# B&R Automation Studio project A2019059_Linka_Power_CP (part 36)

```iecst
            //Polohovanie na pozície skrutiek//
            IF P3_Srobovanie.RR_PolohujNaPoziciuSkrutky_4F5F THEN
                IF P3_Srobovanie.PAR.RR_IndexPozicieSkrutky_4F5F = 0 THEN  //Pozícia skrutky K40 a M5
                    SC_P3_Srobovanie.ResetStep:= TRUE;
                    SC_P3_Srobovanie.Step:= 170;
                ELSIF P3_Srobovanie.PAR.RR_IndexPozicieSkrutky_4F5F = 1 THEN  //Pozícia odobratia skrutky M5
                    SC_P3_Srobovanie.ResetStep:= TRUE;
                    SC_P3_Srobovanie.Step:= 130;
                ELSIF P3_Srobovanie.PAR.RR_IndexPozicieSkrutky_4F5F = 2 THEN  //Pozícia HV testu
                    SC_P3_Srobovanie.ResetStep:= TRUE;
                    SC_P3_Srobovanie.Step:= 300;
                END_IF
            ELSIF P3_Srobovanie.RR_PolohujNaPoziciuSkrutky_5H THEN
                IF P3_Srobovanie.PAR.RR_IndexPozicieSkrutky_5H = 0 THEN  //Pozícia skrutky M5
                    SC_P3_Srobovanie.ResetStep:= TRUE;
                    SC_P3_Srobovanie.Step:= 200;
                ELSIF P3_Srobovanie.PAR.RR_IndexPozicieSkrutky_5H = 1 THEN  //Pozícia odobratia skrutky M5
                    SC_P3_Srobovanie.ResetStep:= TRUE;
                    SC_P3_Srobovanie.Step:= 130;
                ELSIF P3_Srobovanie.PAR.RR_IndexPozicieSkrutky_5H = 2 THEN  //Pozícia HV testu
                    SC_P3_Srobovanie.ResetStep:= TRUE;
                    SC_P3_Srobovanie.Step:= 300;
                END_IF
            END_IF

    END_CASE

END_PROGRAM

PROGRAM _EXIT
	(* Insert code here *)

END_PROGRAM
```

#### Variables.var - Local variables
```iecst
VAR
	Triger_0 : BOOL;
	CasPowerON_OsY : TON;
	SC_OvlManipulatora_OsY : SequenceControlTyp;
	OsY_JoggVPRED : BOOL;
	OsY_JoggVZAD : BOOL;
	OsY_POLOHUJ : BOOL;
	OsY_HOME : BOOL;
	OsY_STOP : BOOL;
	ZadanaPoziciaUINT_OsY : UINT;
	AktualnaPoziciaUINT_OsY : UINT;
	SC_OvlZdvihuHV_Testu : SequenceControlTyp;
	HV_Test_VYSUN : BOOL;
	HV_Test_ZASUN : BOOL;
	SC_OvlKontaktovHV_Testu : SequenceControlTyp;
	Kontakty_VYSUN : BOOL;
	Kontakty_ZASUN : BOOL;
	SC_OvlTesteraHV : SequenceControlTyp;
	SKTcpClientTester_0 : SKTcpClientTester;
	dataStr : STRING[32];
	HV_Test_START : BOOL;
	HV_Test_UKONCENY : BOOL;
	i : USINT;
	CasSrobovania : REAL;
	M5_DosiahnutyMoment_REAL : REAL;
	M5_Moment_ToleranciaMAX_REAL : REAL;
	M5_Moment_ToleranciaMIN_REAL : REAL;
	K40_DosiahnutyMoment_REAL : REAL;
	K40_Moment_ToleranciaMAX_REAL : REAL;
	K40_Moment_ToleranciaMIN_REAL : REAL;
	M5_PrevodMomentu : PrevodMomentu;
	K40_PrevodMomentu : PrevodMomentu;
	CasZastaveniaServa : TON;
	FazaNavratu : UINT;
	CasKontrolyZasobSkrutiek_K40 : TON;
	CasKontrolyZasobSkrutiek_M5 : TON;
	TEST : BOOL;
	PocetDopytovNaTester : USINT;
	SkrutkovanieK40_Ukoncene : BOOL;
	SkrutkovanieM5_Ukoncene : BOOL;
	Skrutkovanie_VysledkyDONE : BOOL;
	PocetVysunutiSkrutkovacky_M5 : USINT;
END_VAR
(******Zápis do ParID serva*************)
VAR
	MC_BR_ProcessParID_AcpAx_0 : MC_BR_ProcessParID_AcpAx := (0);
	McAcpAxProcessParIDType_0 : ARRAY[0..1] OF McAcpAxProcessParIDType;
	OsY_NovaHodnotaMomentu_POS : REAL := 0.0;
	OsY_NovaHodnotaMomentu_NEG : REAL := 0.0;
END_VAR
```

#### OvlManipulatora_OsY.st
```iecst
ACTION OvlManipulatora_OsY:

	//************************Axis 9*******************************//
	//Otáčka serva = 10mm//
	//Motor má absolútny encodér//

    //ENABLE knižnice//
    IF P3_Srobovanie.ServoManipulOsY_M37.STATUS.Communication_READY THEN
        P3_Srobovanie.ServoManipulOsY_M37.CMD.ENABLE:= TRUE;
    ELSE
        P3_Srobovanie.ServoManipulOsY_M37.CMD.ENABLE:= FALSE;
    END_IF

	//Zapnutie serva//
	CasPowerON_OsY.IN:= P3_Srobovanie.ServoManipulOsY_M37.STATUS.ReadyToPower_ON AND P3_Srobovanie.STAV.OsY_LimitSnimace_BUSY AND P3_Srobovanie.ServoManipulOsY_M37.STATUS.EnableSwitch_ACTIVE AND NOT P3_Srobovanie.ServoManipulOsY_M37.STATUS.ERROR;
	IF CasPowerON_OsY.Q THEN
		P3_Srobovanie.ServoManipulOsY_M37.CMD.POWER:= TRUE;
	ELSE
		P3_Srobovanie.ServoManipulOsY_M37.CMD.POWER:= FALSE;
	END_IF

	CasPowerON_OsY.PT:= T#1s;
	CasPowerON_OsY();

	//Reset poruchy//
	IF P3_Srobovanie.ServoManipulOsY_M37.STATUS.ERROR AND P3_Srobovanie.ServoManipulOsY_M37.STATUS.ReadyToPower_ON THEN
		P3_Srobovanie.ServoManipulOsY_M37.CMD.ErrorRESET:= TRUE;
	ELSE
		P3_Srobovanie.ServoManipulOsY_M37.CMD.ErrorRESET:= FALSE;
	END_IF

	//Zobrazenie stavou a parametrov serva//
	P3_Srobovanie.STAV.OsY_AktualnaPozicia:= P3_Srobovanie.ServoManipulOsY_M37.STATUS.ActualPosition;
	P3_Srobovanie.STAV.OsY_AktualnaRychlost:= P3_Srobovanie.ServoManipulOsY_M37.STATUS.ActualVelocity;
	P3_Srobovanie.STAV.OsY_AktualnyMoment:= P3_Srobovanie.ServoManipulOsY_M37.STATUS.ActualTorque;
	P3_Srobovanie.STAV.OsY_HomingOK:= P3_Srobovanie.ServoManipulOsY_M37.STATUS.Homing_OK;
	P3_Srobovanie.STAV.OsY_BUSY:= P3_Srobovanie.ServoManipulOsY_M37.STATUS.MoveAbsolute_BUSY;
	P3_Srobovanie.STAV.OsY_JoggLimitDosiahnuty:= P3_Srobovanie.ServoManipulOsY_M37.STATUS.JoggLimit_Dosiahnuty;

	//Zadané parametre serva//
	P3_Srobovanie.ServoManipulOsY_M37.HomePAR.Acceleration:= 50;
	P3_Srobovanie.ServoManipulOsY_M37.HomePAR.HomingVelocity:= 2;
	P3_Srobovanie.ServoManipulOsY_M37.HomePAR.StartVelocity:= 5;
	P3_Srobovanie.ServoManipulOsY_M37.HomePAR.Position:= -22624.8;    //Offset homing pozície pre absolutny snímač
	P3_Srobovanie.ServoManipulOsY_M37.HomePAR.HomingMode:= 3; //0 - direct, 1- refrenčný snímač, 2 - limitný snímač, 3 - absolutny encoder, 4 - na moment//

	P3_Srobovanie.ServoManipulOsY_M37.PAR.Acceleration:= P34_RemPremenne.P3_ManipSrob_OsY_Rychlost*10;
	P3_Srobovanie.ServoManipulOsY_M37.PAR.Deceleration:= P34_RemPremenne.P3_ManipSrob_OsY_Rychlost*10;
	P3_Srobovanie.ServoManipulOsY_M37.PAR.StopDeceleration:= P34_RemPremenne.P3_ManipSrob_OsY_Rychlost*10;
	P3_Srobovanie.ServoManipulOsY_M37.PAR.Position:= P3_Srobovanie.PAR.OsY_ZadanaPozicia;

	//Zastavenie pohybu serva//
	IF OsY_STOP THEN
		P3_Srobovanie.ServoManipulOsY_M37.CMD.STOP:= TRUE;
		SC_OvlManipulatora_OsY.Step:= 0;
		CasZastaveniaServa.IN:= TRUE;
		OsY_STOP:= FALSE;
	END_IF

	IF CasZastaveniaServa.Q THEN
		P3_Srobovanie.ServoManipulOsY_M37.CMD.STOP:= FALSE;
		CasZastaveniaServa.IN:= FALSE;
	END_IF

	CasZastaveniaServa.PT:= T#2s;
	CasZastaveniaServa();

	//Volanie funkcie SequenceControl//
	SequenceControl(SC:= SC_OvlManipulatora_OsY);

	CASE SC_OvlManipulatora_OsY.Step OF

		0:
			SC_OvlManipulatora_OsY.StepName:= '0 - Nulovanie';
			OsY_JoggVPRED:= FALSE;
			OsY_JoggVZAD:= FALSE;
			OsY_POLOHUJ:= FALSE;
			OsY_HOME:= FALSE;
			P3_Srobovanie.ServoManipulOsY_M37.CMD.HOME:= FALSE;
			P3_Srobovanie.ServoManipulOsY_M37.CMD.JoggVPRED:= FALSE;
			P3_Srobovanie.ServoManipulOsY_M37.CMD.JoggVZAD:= FALSE;
			P3_Srobovanie.ServoManipulOsY_M37.CMD.MoveAbsolute:= FALSE;

			IF SC_P3_Srobovanie.Step <> 0 AND P3_Srobovanie.ServoManipulOsY_M37.STATUS.Power_ON AND NOT P3_Srobovanie.ServoManipulOsY_M37.STATUS.ERROR AND NOT P3_Srobovanie.ServoManipulOsY_M37.STATUS.STOP_ACTIVE THEN
				SC_OvlManipulatora_OsY.ResetStep:= TRUE;
				SC_OvlManipulatora_OsY.Step:= 1;
			END_IF

		1:
			SC_OvlManipulatora_OsY.StepName:= '1 - Rozhodnutie o cinnosti';
			IF OsY_JoggVPRED THEN
				SC_OvlManipulatora_OsY.Step:= 10;
			ELSIF OsY_JoggVZAD THEN
				SC_OvlManipulatora_OsY.Step:= 20;
			ELSIF OsY_HOME THEN
				SC_OvlManipulatora_OsY.Step:= 30;
			ELSIF OsY_POLOHUJ THEN
				SC_OvlManipulatora_OsY.Step:= 40;
			END_IF

		10:
			SC_OvlManipulatora_OsY.StepName:= '10 - Jogg VPRED';
			SC_OvlManipulatora_OsY.IdleTime.PT:= T#3s;
			SC_OvlManipulatora_OsY.AlarmTime.PT:= T#3s;

			IF NOT SC_OvlManipulatora_OsY.Switch1 THEN
				P3_Srobovanie.ServoManipulOsY_M37.CMD.JoggVPRED:= TRUE;
				SC_OvlManipulatora_OsY.Switch1:= TRUE;
			END_IF

			IF NOT OsY_JoggVPRED THEN
				SC_OvlManipulatora_OsY.ResetStep:= TRUE;
				SC_OvlManipulatora_OsY.Step:= 0;
			END_IF

		20:
			SC_OvlManipulatora_OsY.StepName:= '20 - Jogg VZAD';
			SC_OvlManipulatora_OsY.IdleTime.PT:= T#3s;
			SC_OvlManipulatora_OsY.AlarmTime.PT:= T#3s;

			IF NOT SC_OvlManipulatora_OsY.Switch1 THEN
				P3_Srobovanie.ServoManipulOsY_M37.CMD.JoggVZAD:= TRUE;
				SC_OvlManipulatora_OsY.Switch1:= TRUE;
			END_IF

			IF NOT OsY_JoggVZAD THEN
				SC_OvlManipulatora_OsY.ResetStep:= TRUE;
				SC_OvlManipulatora_OsY.Step:= 0;
			END_IF

		30:
			SC_OvlManipulatora_OsY.StepName:= '30 - Homing';
			SC_OvlManipulatora_OsY.IdleTime.PT:= T#500ms;
			SC_OvlManipulatora_OsY.AlarmTime.PT:= T#3s;

			IF NOT SC_OvlManipulatora_OsY.Switch1 THEN
				P3_Srobovanie.ServoManipulOsY_M37.CMD.HOME:= TRUE;
				SC_OvlManipulatora_OsY.IdleTime.IN:= TRUE;
				SC_OvlManipulatora_OsY.Switch1:= TRUE;
			END_IF

			IF P3_Srobovanie.ServoManipulOsY_M37.STATUS.Homing_OK AND SC_OvlManipulatora_OsY.IdleTime.Q THEN
				SC_OvlManipulatora_OsY.ResetStep:= TRUE;
				SC_OvlManipulatora_OsY.Step:= 0;
			END_IF

		40:
			SC_OvlManipulatora_OsY.StepName:= '40 - Polohovanie';
			SC_OvlManipulatora_OsY.IdleTime.PT:= T#500ms;
			SC_OvlManipulatora_OsY.AlarmTime.PT:= T#3s;

			ZadanaPoziciaUINT_OsY:= LREAL_TO_UINT(P3_Srobovanie.PAR.OsY_ZadanaPozicia);
			AktualnaPoziciaUINT_OsY:= LREAL_TO_UINT(P3_Srobovanie.STAV.OsY_AktualnaPozicia);

			IF NOT SC_OvlManipulatora_OsY.Switch1 THEN
				P3_Srobovanie.ServoManipulOsY_M37.CMD.MoveAbsolute:= TRUE;
				SC_OvlManipulatora_OsY.Switch1:= TRUE;
			END_IF

			IF (AktualnaPoziciaUINT_OsY = ZadanaPoziciaUINT_OsY) AND P3_Srobovanie.ServoManipulOsY_M37.STATUS.MoveAbsolute_DONE THEN
				P3_Srobovanie.STAV.OsY_PoziciaDosiahnuta:= TRUE;
				SC_OvlManipulatora_OsY.ResetStep:= TRUE;
				SC_OvlManipulatora_OsY.Step:= 0;
			END_IF

	END_CASE

END_ACTION
```

#### AtlasCopcoKomunikacia.st
```iecst
ACTION AtlasCopcoKomunikacia:

    M5_PrevodMomentu();
    K40_PrevodMomentu();

	//**************************************************************Skrutkovacka M5**************************************************************//
	//Vstupy z AtlasCopco do PLC//
    P3_Srobovanie.Skrutkovacka_M5.Stav_VysledokPotvrdeny:= P3_Srobovanie.PAR.M5_AtlasCopcoInputs[0].0;
    P3_Srobovanie.Skrutkovacka_M5.Stav_EmergencyStop:= P3_Srobovanie.PAR.M5_AtlasCopcoInputs[0].1;
    P3_Srobovanie.Skrutkovacka_M5.Stav_READY_to_START:= P3_Srobovanie.PAR.M5_AtlasCopcoInputs[0].2;
    P3_Srobovanie.Skrutkovacka_M5.Stav_MANUAL:= P3_Srobovanie.PAR.M5_AtlasCopcoInputs[0].3;
    P3_Srobovanie.Skrutkovacka_M5.Stav_UtahovanieUkoncene:= P3_Srobovanie.PAR.M5_AtlasCopcoInputs[0].4;
    P3_Srobovanie.Skrutkovacka_M5.Stav_VysledokUtahovania_NG:= P3_Srobovanie.PAR.M5_AtlasCopcoInputs[0].5;
    P3_Srobovanie.Skrutkovacka_M5.Stav_VysledokUtahovania_OK:= P3_Srobovanie.PAR.M5_AtlasCopcoInputs[0].6;
    P3_Srobovanie.Skrutkovacka_M5.Stav_SmerOtacania_VPRED:= P3_Srobovanie.PAR.M5_AtlasCopcoInputs[0].7;
    P3_Srobovanie.Skrutkovacka_M5.Stav_BUSY:= P3_Srobovanie.PAR.M5_AtlasCopcoInputs[0].8;
    P3_Srobovanie.Skrutkovacka_M5.Stav_ControlerSwitch_ON:= P3_Srobovanie.PAR.M5_AtlasCopcoInputs[0].9;
    P3_Srobovanie.Skrutkovacka_M5.Stav_Station_READY:= P3_Srobovanie.PAR.M5_AtlasCopcoInputs[0].10;
    P3_Srobovanie.Skrutkovacka_M5.Stav_NastrojPripojeny:= P3_Srobovanie.PAR.M5_AtlasCopcoInputs[0].11;
    P3_Srobovanie.Skrutkovacka_M5.Stav_NastrojUtahuje:= P3_Srobovanie.PAR.M5_AtlasCopcoInputs[0].12;

    //Výstupy z PLC do AtlasCopco//
    P3_Srobovanie.PAR.M5_AllasCopcoOutputs[0].0:= P3_Srobovanie.Skrutkovacka_M5.RESET_Poruchy;
    P3_Srobovanie.PAR.M5_AllasCopcoOutputs[0].1:= P3_Srobovanie.Skrutkovacka_M5.RESET_Vysledkov;
    P3_Srobovanie.PAR.M5_AllasCopcoOutputs[0].2:= P3_Srobovanie.Skrutkovacka_M5.START_Skrutkovania;
    P3_Srobovanie.PAR.M5_AllasCopcoOutputs[0].3:= P3_Srobovanie.Skrutkovacka_M5.START_Utahovania;

    //Dosiahnutý moment//
//    P3_Srobovanie.STAV.M5_DosiahnutyMoment.0:= P3_Srobovanie.PAR.M5_AtlasCopcoInputs[1].24;
//    P3_Srobovanie.STAV.M5_DosiahnutyMoment.1:= P3_Srobovanie.PAR.M5_AtlasCopcoInputs[1].25;
//    P3_Srobovanie.STAV.M5_DosiahnutyMoment.2:= P3_Srobovanie.PAR.M5_AtlasCopcoInputs[1].26;
//    P3_Srobovanie.STAV.M5_DosiahnutyMoment.3:= P3_Srobovanie.PAR.M5_AtlasCopcoInputs[1].27;
//    P3_Srobovanie.STAV.M5_DosiahnutyMoment.4:= P3_Srobovanie.PAR.M5_AtlasCopcoInputs[1].28;
//    P3_Srobovanie.STAV.M5_DosiahnutyMoment.5:= P3_Srobovanie.PAR.M5_AtlasCopcoInputs[1].29;
//    P3_Srobovanie.STAV.M5_DosiahnutyMoment.6:= P3_Srobovanie.PAR.M5_AtlasCopcoInputs[1].30;
//    P3_Srobovanie.STAV.M5_DosiahnutyMoment.7:= P3_Srobovanie.PAR.M5_AtlasCopcoInputs[1].31;
//    P3_Srobovanie.STAV.M5_DosiahnutyMoment.8:= P3_Srobovanie.PAR.M5_AtlasCopcoInputs[1].16;
//    P3_Srobovanie.STAV.M5_DosiahnutyMoment.9:= P3_Srobovanie.PAR.M5_AtlasCopcoInputs[1].17;
//    P3_Srobovanie.STAV.M5_DosiahnutyMoment.10:= P3_Srobovanie.PAR.M5_AtlasCopcoInputs[1].18;
//    P3_Srobovanie.STAV.M5_DosiahnutyMoment.11:= P3_Srobovanie.PAR.M5_AtlasCopcoInputs[1].19;
//    P3_Srobovanie.STAV.M5_DosiahnutyMoment.12:= P3_Srobovanie.PAR.M5_AtlasCopcoInputs[1].20;
//    P3_Srobovanie.STAV.M5_DosiahnutyMoment.13:= P3_Srobovanie.PAR.M5_AtlasCopcoInputs[1].21;
//    P3_Srobovanie.STAV.M5_DosiahnutyMoment.14:= P3_Srobovanie.PAR.M5_AtlasCopcoInputs[1].22;
//    P3_Srobovanie.STAV.M5_DosiahnutyMoment.15:= P3_Srobovanie.PAR.M5_AtlasCopcoInputs[1].23;
//    P3_Srobovanie.STAV.M5_DosiahnutyMoment.16:= P3_Srobovanie.PAR.M5_AtlasCopcoInputs[1].8;
//    P3_Srobovanie.STAV.M5_DosiahnutyMoment.17:= P3_Srobovanie.PAR.M5_AtlasCopcoInputs[1].9;
//    P3_Srobovanie.STAV.M5_DosiahnutyMoment.18:= P3_Srobovanie.PAR.M5_AtlasCopcoInputs[1].10;
//    P3_Srobovanie.STAV.M5_DosiahnutyMoment.19:= P3_Srobovanie.PAR.M5_AtlasCopcoInputs[1].11;
//    P3_Srobovanie.STAV.M5_DosiahnutyMoment.20:= P3_Srobovanie.PAR.M5_AtlasCopcoInputs[1].12;
//    P3_Srobovanie.STAV.M5_DosiahnutyMoment.21:= P3_Srobovanie.PAR.M5_AtlasCopcoInputs[1].13;
//    P3_Srobovanie.STAV.M5_DosiahnutyMoment.22:= P3_Srobovanie.PAR.M5_AtlasCopcoInputs[1].14;
//    P3_Srobovanie.STAV.M5_DosiahnutyMoment.23:= P3_Srobovanie.PAR.M5_AtlasCopcoInputs[1].15;
//    P3_Srobovanie.STAV.M5_DosiahnutyMoment.24:= P3_Srobovanie.PAR.M5_AtlasCopcoInputs[1].0;
//    P3_Srobovanie.STAV.M5_DosiahnutyMoment.25:= P3_Srobovanie.PAR.M5_AtlasCopcoInputs[1].1;
//    P3_Srobovanie.STAV.M5_DosiahnutyMoment.26:= P3_Srobovanie.PAR.M5_AtlasCopcoInputs[1].2;
//    P3_Srobovanie.STAV.M5_DosiahnutyMoment.27:= P3_Srobovanie.PAR.M5_AtlasCopcoInputs[1].3;
//    P3_Srobovanie.STAV.M5_DosiahnutyMoment.28:= P3_Srobovanie.PAR.M5_AtlasCopcoInputs[1].4;
//    P3_Srobovanie.STAV.M5_DosiahnutyMoment.29:= P3_Srobovanie.PAR.M5_AtlasCopcoInputs[1].5;
//    P3_Srobovanie.STAV.M5_DosiahnutyMoment.30:= P3_Srobovanie.PAR.M5_AtlasCopcoInputs[1].6;
//    P3_Srobovanie.STAV.M5_DosiahnutyMoment.31:= P3_Srobovanie.PAR.M5_AtlasCopcoInputs[1].7;
//    M5_DosiahnutyMoment_REAL:= UDINT_TO_REAL(P3_Srobovanie.STAV.M5_DosiahnutyMoment);
//    IF M5_DosiahnutyMoment_REAL > 0 THEN
//       P3_Srobovanie.STAV.M5_DosiahnutyMoment_REAL:= (M5_DosiahnutyMoment_REAL*2.34)/131106;
//    ELSE
//        P3_Srobovanie.STAV.M5_DosiahnutyMoment_REAL:= 0.0;
//    END_IF

    M5_PrevodMomentu.AtlasAktualnyMoment:=P3_Srobovanie.PAR.M5_AtlasCopcoInputs[1];
    P3_Srobovanie.STAV.M5_DosiahnutyMoment_REAL:=M5_PrevodMomentu.AktualnyMoment;

    (*P3_Srobovanie.STAV.M5_DosiahnutyMoment_REAL:= M5_DosiahnutyMoment_REAL /100;*)

    //Moment - Tolerancia MAX//
//    P3_Srobovanie.STAV.M5_Moment_ToleranciaMAX.0:= P3_Srobovanie.PAR.M5_AtlasCopcoInputs[3].24;
//    P3_Srobovanie.STAV.M5_Moment_ToleranciaMAX.1:= P3_Srobovanie.PAR.M5_AtlasCopcoInputs[3].25;
//    P3_Srobovanie.STAV.M5_Moment_ToleranciaMAX.2:= P3_Srobovanie.PAR.M5_AtlasCopcoInputs[3].26;
//    P3_Srobovanie.STAV.M5_Moment_ToleranciaMAX.3:= P3_Srobovanie.PAR.M5_AtlasCopcoInputs[3].27;
//    P3_Srobovanie.STAV.M5_Moment_ToleranciaMAX.4:= P3_Srobovanie.PAR.M5_AtlasCopcoInputs[3].28;
//    P3_Srobovanie.STAV.M5_Moment_ToleranciaMAX.5:= P3_Srobovanie.PAR.M5_AtlasCopcoInputs[3].29;
//    P3_Srobovanie.STAV.M5_Moment_ToleranciaMAX.6:= P3_Srobovanie.PAR.M5_AtlasCopcoInputs[3].30;
//    P3_Srobovanie.STAV.M5_Moment_ToleranciaMAX.7:= P3_Srobovanie.PAR.M5_AtlasCopcoInputs[3].31;
//    P3_Srobovanie.STAV.M5_Moment_ToleranciaMAX.8:= P3_Srobovanie.PAR.M5_AtlasCopcoInputs[3].16;
//    P3_Srobovanie.STAV.M5_Moment_ToleranciaMAX.9:= P3_Srobovanie.PAR.M5_AtlasCopcoInputs[3].17;
//    P3_Srobovanie.STAV.M5_Moment_ToleranciaMAX.10:= P3_Srobovanie.PAR.M5_AtlasCopcoInputs[3].18;
//    P3_Srobovanie.STAV.M5_Moment_ToleranciaMAX.11:= P3_Srobovanie.PAR.M5_AtlasCopcoInputs[3].19;
//    P3_Srobovanie.STAV.M5_Moment_ToleranciaMAX.12:= P3_Srobovanie.PAR.M5_AtlasCopcoInputs[3].20;
//    P3_Srobovanie.STAV.M5_Moment_ToleranciaMAX.13:= P3_Srobovanie.PAR.M5_AtlasCopcoInputs[3].21;
//    P3_Srobovanie.STAV.M5_Moment_ToleranciaMAX.14:= P3_Srobovanie.PAR.M5_AtlasCopcoInputs[3].22;
//    P3_Srobovanie.STAV.M5_Moment_ToleranciaMAX.15:= P3_Srobovanie.PAR.M5_AtlasCopcoInputs[3].23;
//    P3_Srobovanie.STAV.M5_Moment_ToleranciaMAX.16:= P3_Srobovanie.PAR.M5_AtlasCopcoInputs[3].8;
//    P3_Srobovanie.STAV.M5_Moment_ToleranciaMAX.17:= P3_Srobovanie.PAR.M5_AtlasCopcoInputs[3].9;
//    P3_Srobovanie.STAV.M5_Moment_ToleranciaMAX.18:= P3_Srobovanie.PAR.M5_AtlasCopcoInputs[3].10;
//    P3_Srobovanie.STAV.M5_Moment_ToleranciaMAX.19:= P3_Srobovanie.PAR.M5_AtlasCopcoInputs[3].11;
//    P3_Srobovanie.STAV.M5_Moment_ToleranciaMAX.20:= P3_Srobovanie.PAR.M5_AtlasCopcoInputs[3].12;
//    P3_Srobovanie.STAV.M5_Moment_ToleranciaMAX.21:= P3_Srobovanie.PAR.M5_AtlasCopcoInputs[3].13;
//    P3_Srobovanie.STAV.M5_Moment_ToleranciaMAX.22:= P3_Srobovanie.PAR.M5_AtlasCopcoInputs[3].14;
//    P3_Srobovanie.STAV.M5_Moment_ToleranciaMAX.23:= P3_Srobovanie.PAR.M5_AtlasCopcoInputs[3].15;
//    P3_Srobovanie.STAV.M5_Moment_ToleranciaMAX.24:= P3_Srobovanie.PAR.M5_AtlasCopcoInputs[3].0;
//    P3_Srobovanie.STAV.M5_Moment_ToleranciaMAX.25:= P3_Srobovanie.PAR.M5_AtlasCopcoInputs[3].1;
//    P3_Srobovanie.STAV.M5_Moment_ToleranciaMAX.26:= P3_Srobovanie.PAR.M5_AtlasCopcoInputs[3].2;
//    P3_Srobovanie.STAV.M5_Moment_ToleranciaMAX.27:= P3_Srobovanie.PAR.M5_AtlasCopcoInputs[3].3;
//    P3_Srobovanie.STAV.M5_Moment_ToleranciaMAX.28:= P3_Srobovanie.PAR.M5_AtlasCopcoInputs[3].4;
//    P3_Srobovanie.STAV.M5_Moment_ToleranciaMAX.29:= P3_Srobovanie.PAR.M5_AtlasCopcoInputs[3].5;
//    P3_Srobovanie.STAV.M5_Moment_ToleranciaMAX.30:= P3_Srobovanie.PAR.M5_AtlasCopcoInputs[3].6;
//    P3_Srobovanie.STAV.M5_Moment_ToleranciaMAX.31:= P3_Srobovanie.PAR.M5_AtlasCopcoInputs[3].7;
//    M5_Moment_ToleranciaMAX_REAL:= UDINT_TO_REAL(P3_Srobovanie.STAV.M5_Moment_ToleranciaMAX);
//    IF M5_Moment_ToleranciaMAX_REAL > 0 THEN
//      P3_Srobovanie.STAV.M5_Moment_ToleranciaMAX_REAL:= (M5_Moment_ToleranciaMAX_REAL*2.82)/131154;
//    ELSE
//        P3_Srobovanie.STAV.M5_Moment_ToleranciaMAX_REAL:= 0.0;
//    END_IF
//

    M5_PrevodMomentu.AtlasMaximalnaTolerancia:=P3_Srobovanie.PAR.M5_AtlasCopcoInputs[3];
    P3_Srobovanie.STAV.M5_Moment_ToleranciaMAX_REAL:=M5_PrevodMomentu.ToleranciaMAX;

    (*P3_Srobovanie.STAV.M5_Moment_ToleranciaMAX_REAL:= M5_Moment_ToleranciaMAX_REAL /100;*)

    //Moment - Tolerancia MIN//
//    P3_Srobovanie.STAV.M5_Moment_ToleranciaMIN.0:= P3_Srobovanie.PAR.M5_AtlasCopcoInputs[4].24;
//    P3_Srobovanie.STAV.M5_Moment_ToleranciaMIN.1:= P3_Srobovanie.PAR.M5_AtlasCopcoInputs[4].25;
//    P3_Srobovanie.STAV.M5_Moment_ToleranciaMIN.2:= P3_Srobovanie.PAR.M5_AtlasCopcoInputs[4].26;
//    P3_Srobovanie.STAV.M5_Moment_ToleranciaMIN.3:= P3_Srobovanie.PAR.M5_AtlasCopcoInputs[4].27;
//    P3_Srobovanie.STAV.M5_Moment_ToleranciaMIN.4:= P3_Srobovanie.PAR.M5_AtlasCopcoInputs[4].28;
//    P3_Srobovanie.STAV.M5_Moment_ToleranciaMIN.5:= P3_Srobovanie.PAR.M5_AtlasCopcoInputs[4].29;
//    P3_Srobovanie.STAV.M5_Moment_ToleranciaMIN.6:= P3_Srobovanie.PAR.M5_AtlasCopcoInputs[4].30;
//    P3_Srobovanie.STAV.M5_Moment_ToleranciaMIN.7:= P3_Srobovanie.PAR.M5_AtlasCopcoInputs[4].31;
//    P3_Srobovanie.STAV.M5_Moment_ToleranciaMIN.8:= P3_Srobovanie.PAR.M5_AtlasCopcoInputs[4].16;
//    P3_Srobovanie.STAV.M5_Moment_ToleranciaMIN.9:= P3_Srobovanie.PAR.M5_AtlasCopcoInputs[4].17;
//    P3_Srobovanie.STAV.M5_Moment_ToleranciaMIN.10:= P3_Srobovanie.PAR.M5_AtlasCopcoInputs[4].18;
//    P3_Srobovanie.STAV.M5_Moment_ToleranciaMIN.11:= P3_Srobovanie.PAR.M5_AtlasCopcoInputs[4].19;
//    P3_Srobovanie.STAV.M5_Moment_ToleranciaMIN.12:= P3_Srobovanie.PAR.M5_AtlasCopcoInputs[4].20;
//    P3_Srobovanie.STAV.M5_Moment_ToleranciaMIN.13:= P3_Srobovanie.PAR.M5_AtlasCopcoInputs[4].21;
//    P3_Srobovanie.STAV.M5_Moment_ToleranciaMIN.14:= P3_Srobovanie.PAR.M5_AtlasCopcoInputs[4].22;
//    P3_Srobovanie.STAV.M5_Moment_ToleranciaMIN.15:= P3_Srobovanie.PAR.M5_AtlasCopcoInputs[4].23;
//    P3_Srobovanie.STAV.M5_Moment_ToleranciaMIN.16:= P3_Srobovanie.PAR.M5_AtlasCopcoInputs[4].8;
//    P3_Srobovanie.STAV.M5_Moment_ToleranciaMIN.17:= P3_Srobovanie.PAR.M5_AtlasCopcoInputs[4].9;
//    P3_Srobovanie.STAV.M5_Moment_ToleranciaMIN.18:= P3_Srobovanie.PAR.M5_AtlasCopcoInputs[4].10;
//    P3_Srobovanie.STAV.M5_Moment_ToleranciaMIN.19:= P3_Srobovanie.PAR.M5_AtlasCopcoInputs[4].11;
//    P3_Srobovanie.STAV.M5_Moment_ToleranciaMIN.20:= P3_Srobovanie.PAR.M5_AtlasCopcoInputs[4].12;
//    P3_Srobovanie.STAV.M5_Moment_ToleranciaMIN.21:= P3_Srobovanie.PAR.M5_AtlasCopcoInputs[4].13;
//    P3_Srobovanie.STAV.M5_Moment_ToleranciaMIN.22:= P3_Srobovanie.PAR.M5_AtlasCopcoInputs[4].14;
//    P3_Srobovanie.STAV.M5_Moment_ToleranciaMIN.23:= P3_Srobovanie.PAR.M5_AtlasCopcoInputs[4].15;
//    P3_Srobovanie.STAV.M5_Moment_ToleranciaMIN.24:= P3_Srobovanie.PAR.M5_AtlasCopcoInputs[4].0;
//    P3_Srobovanie.STAV.M5_Moment_ToleranciaMIN.25:= P3_Srobovanie.PAR.M5_AtlasCopcoInputs[4].1;
//    P3_Srobovanie.STAV.M5_Moment_ToleranciaMIN.26:= P3_Srobovanie.PAR.M5_AtlasCopcoInputs[4].2;
//    P3_Srobovanie.STAV.M5_Moment_ToleranciaMIN.27:= P3_Srobovanie.PAR.M5_AtlasCopcoInputs[4].3;
//    P3_Srobovanie.STAV.M5_Moment_ToleranciaMIN.28:= P3_Srobovanie.PAR.M5_AtlasCopcoInputs[4].4;
//    P3_Srobovanie.STAV.M5_Moment_ToleranciaMIN.29:= P3_Srobovanie.PAR.M5_AtlasCopcoInputs[4].5;
//    P3_Srobovanie.STAV.M5_Moment_ToleranciaMIN.30:= P3_Srobovanie.PAR.M5_AtlasCopcoInputs[4].6;
//    P3_Srobovanie.STAV.M5_Moment_ToleranciaMIN.31:= P3_Srobovanie.PAR.M5_AtlasCopcoInputs[4].7;
//    M5_Moment_ToleranciaMIN_REAL:= UDINT_TO_REAL(P3_Srobovanie.STAV.M5_Moment_ToleranciaMIN);
//    IF M5_Moment_ToleranciaMIN_REAL > 0 THEN
//       P3_Srobovanie.STAV.M5_Moment_ToleranciaMIN_REAL:= (M5_Moment_ToleranciaMIN_REAL*2.34)/131106;
//    ELSE
//        P3_Srobovanie.STAV.M5_Moment_ToleranciaMIN_REAL:= 0.0;
//    END_IF

    M5_PrevodMomentu.AtlasMinimalnaTolerancia:=P3_Srobovanie.PAR.M5_AtlasCopcoInputs[4];
    P3_Srobovanie.STAV.M5_Moment_ToleranciaMIN_REAL:=M5_PrevodMomentu.ToleranciaMIN;

    (*P3_Srobovanie.STAV.M5_Moment_ToleranciaMIN_REAL:= M5_Moment_ToleranciaMIN_REAL/100;*)

    //Dosiahnutý úhol//
    P3_Srobovanie.STAV.M5_DosiahnutyUhol.0:= P3_Srobovanie.PAR.M5_AtlasCopcoInputs[0].24;
    P3_Srobovanie.STAV.M5_DosiahnutyUhol.1:= P3_Srobovanie.PAR.M5_AtlasCopcoInputs[0].25;
    P3_Srobovanie.STAV.M5_DosiahnutyUhol.2:= P3_Srobovanie.PAR.M5_AtlasCopcoInputs[0].26;
    P3_Srobovanie.STAV.M5_DosiahnutyUhol.3:= P3_Srobovanie.PAR.M5_AtlasCopcoInputs[0].27;
    P3_Srobovanie.STAV.M5_DosiahnutyUhol.4:= P3_Srobovanie.PAR.M5_AtlasCopcoInputs[0].28;
    P3_Srobovanie.STAV.M5_DosiahnutyUhol.5:= P3_Srobovanie.PAR.M5_AtlasCopcoInputs[0].29;
    P3_Srobovanie.STAV.M5_DosiahnutyUhol.6:= P3_Srobovanie.PAR.M5_AtlasCopcoInputs[0].30;
    P3_Srobovanie.STAV.M5_DosiahnutyUhol.7:= P3_Srobovanie.PAR.M5_AtlasCopcoInputs[0].31;
    P3_Srobovanie.STAV.M5_DosiahnutyUhol.8:= P3_Srobovanie.PAR.M5_AtlasCopcoInputs[0].16;
    P3_Srobovanie.STAV.M5_DosiahnutyUhol.9:= P3_Srobovanie.PAR.M5_AtlasCopcoInputs[0].17;
    P3_Srobovanie.STAV.M5_DosiahnutyUhol.10:= P3_Srobovanie.PAR.M5_AtlasCopcoInputs[0].18;
    P3_Srobovanie.STAV.M5_DosiahnutyUhol.11:= P3_Srobovanie.PAR.M5_AtlasCopcoInputs[0].19;
    P3_Srobovanie.STAV.M5_DosiahnutyUhol.12:= P3_Srobovanie.PAR.M5_AtlasCopcoInputs[0].20;
    P3_Srobovanie.STAV.M5_DosiahnutyUhol.13:= P3_Srobovanie.PAR.M5_AtlasCopcoInputs[0].21;
    P3_Srobovanie.STAV.M5_DosiahnutyUhol.14:= P3_Srobovanie.PAR.M5_AtlasCopcoInputs[0].22;
    P3_Srobovanie.STAV.M5_DosiahnutyUhol.15:= P3_Srobovanie.PAR.M5_AtlasCopcoInputs[0].23;

    //Uhol - Tolerancia MAX//
    P3_Srobovanie.STAV.M5_Uhol_ToleranciaMAX.0:= P3_Srobovanie.PAR.M5_AtlasCopcoInputs[2].8;
    P3_Srobovanie.STAV.M5_Uhol_ToleranciaMAX.1:= P3_Srobovanie.PAR.M5_AtlasCopcoInputs[2].9;
    P3_Srobovanie.STAV.M5_Uhol_ToleranciaMAX.2:= P3_Srobovanie.PAR.M5_AtlasCopcoInputs[2].10;
    P3_Srobovanie.STAV.M5_Uhol_ToleranciaMAX.3:= P3_Srobovanie.PAR.M5_AtlasCopcoInputs[2].11;
    P3_Srobovanie.STAV.M5_Uhol_ToleranciaMAX.4:= P3_Srobovanie.PAR.M5_AtlasCopcoInputs[2].12;
    P3_Srobovanie.STAV.M5_Uhol_ToleranciaMAX.5:= P3_Srobovanie.PAR.M5_AtlasCopcoInputs[2].13;
    P3_Srobovanie.STAV.M5_Uhol_ToleranciaMAX.6:= P3_Srobovanie.PAR.M5_AtlasCopcoInputs[2].14;
    P3_Srobovanie.STAV.M5_Uhol_ToleranciaMAX.7:= P3_Srobovanie.PAR.M5_AtlasCopcoInputs[2].15;
    P3_Srobovanie.STAV.M5_Uhol_ToleranciaMAX.8:= P3_Srobovanie.PAR.M5_AtlasCopcoInputs[2].0;
    P3_Srobovanie.STAV.M5_Uhol_ToleranciaMAX.9:= P3_Srobovanie.PAR.M5_AtlasCopcoInputs[2].1;
    P3_Srobovanie.STAV.M5_Uhol_ToleranciaMAX.10:= P3_Srobovanie.PAR.M5_AtlasCopcoInputs[2].2;
    P3_Srobovanie.STAV.M5_Uhol_ToleranciaMAX.11:= P3_Srobovanie.PAR.M5_AtlasCopcoInputs[2].3;
    P3_Srobovanie.STAV.M5_Uhol_ToleranciaMAX.12:= P3_Srobovanie.PAR.M5_AtlasCopcoInputs[2].4;
    P3_Srobovanie.STAV.M5_Uhol_ToleranciaMAX.13:= P3_Srobovanie.PAR.M5_AtlasCopcoInputs[2].5;
    P3_Srobovanie.STAV.M5_Uhol_ToleranciaMAX.14:= P3_Srobovanie.PAR.M5_AtlasCopcoInputs[2].6;
    P3_Srobovanie.STAV.M5_Uhol_ToleranciaMAX.15:= P3_Srobovanie.PAR.M5_AtlasCopcoInputs[2].7;

    //Uhol - Tolerancia MIN//
    P3_Srobovanie.STAV.M5_Uhol_ToleranciaMIN.0:= P3_Srobovanie.PAR.M5_AtlasCopcoInputs[2].24;
    P3_Srobovanie.STAV.M5_Uhol_ToleranciaMIN.1:= P3_Srobovanie.PAR.M5_AtlasCopcoInputs[2].25;
    P3_Srobovanie.STAV.M5_Uhol_ToleranciaMIN.2:= P3_Srobovanie.PAR.M5_AtlasCopcoInputs[2].26;
    P3_Srobovanie.STAV.M5_Uhol_ToleranciaMIN.3:= P3_Srobovanie.PAR.M5_AtlasCopcoInputs[2].27;
    P3_Srobovanie.STAV.M5_Uhol_ToleranciaMIN.4:= P3_Srobovanie.PAR.M5_AtlasCopcoInputs[2].28;
    P3_Srobovanie.STAV.M5_Uhol_ToleranciaMIN.5:= P3_Srobovanie.PAR.M5_AtlasCopcoInputs[2].29;
    P3_Srobovanie.STAV.M5_Uhol_ToleranciaMIN.6:= P3_Srobovanie.PAR.M5_AtlasCopcoInputs[2].30;
    P3_Srobovanie.STAV.M5_Uhol_ToleranciaMIN.7:= P3_Srobovanie.PAR.M5_AtlasCopcoInputs[2].31;
    P3_Srobovanie.STAV.M5_Uhol_ToleranciaMIN.8:= P3_Srobovanie.PAR.M5_AtlasCopcoInputs[2].16;
    P3_Srobovanie.STAV.M5_Uhol_ToleranciaMIN.9:= P3_Srobovanie.PAR.M5_AtlasCopcoInputs[2].17;
    P3_Srobovanie.STAV.M5_Uhol_ToleranciaMIN.10:= P3_Srobovanie.PAR.M5_AtlasCopcoInputs[2].18;
    P3_Srobovanie.STAV.M5_Uhol_ToleranciaMIN.11:= P3_Srobovanie.PAR.M5_AtlasCopcoInputs[2].19;
    P3_Srobovanie.STAV.M5_Uhol_ToleranciaMIN.12:= P3_Srobovanie.PAR.M5_AtlasCopcoInputs[2].20;
    P3_Srobovanie.STAV.M5_Uhol_ToleranciaMIN.13:= P3_Srobovanie.PAR.M5_AtlasCopcoInputs[2].21;
    P3_Srobovanie.STAV.M5_Uhol_ToleranciaMIN.14:= P3_Srobovanie.PAR.M5_AtlasCopcoInputs[2].22;
    P3_Srobovanie.STAV.M5_Uhol_ToleranciaMIN.15:= P3_Srobovanie.PAR.M5_AtlasCopcoInputs[2].23;

    //***********************************************Skrutkovacka K40**********************************************************************//
    //Vstupy z AtlasCopco do PLC//
    P3_Srobovanie.Skrutkovacka_K40.Stav_VysledokPotvrdeny:= P3_Srobovanie.PAR.K40_AtlasCopcoInputs[0].0;
    P3_Srobovanie.Skrutkovacka_K40.Stav_EmergencyStop:= P3_Srobovanie.PAR.K40_AtlasCopcoInputs[0].1;
    P3_Srobovanie.Skrutkovacka_K40.Stav_READY_to_START:= P3_Srobovanie.PAR.K40_AtlasCopcoInputs[0].2;
    P3_Srobovanie.Skrutkovacka_K40.Stav_MANUAL:= P3_Srobovanie.PAR.K40_AtlasCopcoInputs[0].3;
    P3_Srobovanie.Skrutkovacka_K40.Stav_UtahovanieUkoncene:= P3_Srobovanie.PAR.K40_AtlasCopcoInputs[0].4;
    P3_Srobovanie.Skrutkovacka_K40.Stav_VysledokUtahovania_NG:= P3_Srobovanie.PAR.K40_AtlasCopcoInputs[0].5;
    P3_Srobovanie.Skrutkovacka_K40.Stav_VysledokUtahovania_OK:= P3_Srobovanie.PAR.K40_AtlasCopcoInputs[0].6;
    P3_Srobovanie.Skrutkovacka_K40.Stav_SmerOtacania_VPRED:= P3_Srobovanie.PAR.K40_AtlasCopcoInputs[0].7;
    P3_Srobovanie.Skrutkovacka_K40.Stav_BUSY:= P3_Srobovanie.PAR.K40_AtlasCopcoInputs[0].8;
    P3_Srobovanie.Skrutkovacka_K40.Stav_ControlerSwitch_ON:= P3_Srobovanie.PAR.K40_AtlasCopcoInputs[0].9;
    P3_Srobovanie.Skrutkovacka_K40.Stav_Station_READY:= P3_Srobovanie.PAR.K40_AtlasCopcoInputs[0].10;
    P3_Srobovanie.Skrutkovacka_K40.Stav_NastrojPripojeny:= P3_Srobovanie.PAR.K40_AtlasCopcoInputs[0].11;
    P3_Srobovanie.Skrutkovacka_K40.Stav_NastrojUtahuje:= P3_Srobovanie.PAR.K40_AtlasCopcoInputs[0].12;

    //Výstupy z PLC do AtlasCopco//
    P3_Srobovanie.PAR.K40_AllasCopcoOutputs[0].0:= P3_Srobovanie.Skrutkovacka_K40.RESET_Poruchy;
    P3_Srobovanie.PAR.K40_AllasCopcoOutputs[0].1:= P3_Srobovanie.Skrutkovacka_K40.RESET_Vysledkov;
    P3_Srobovanie.PAR.K40_AllasCopcoOutputs[0].2:= P3_Srobovanie.Skrutkovacka_K40.START_Skrutkovania;
    P3_Srobovanie.PAR.K40_AllasCopcoOutputs[0].3:= P3_Srobovanie.Skrutkovacka_K40.START_Utahovania;

    //Dosiahnutý moment//
//    P3_Srobovanie.STAV.K40_DosiahnutyMoment.0:= P3_Srobovanie.PAR.K40_AtlasCopcoInputs[1].24;
//    P3_Srobovanie.STAV.K40_DosiahnutyMoment.1:= P3_Srobovanie.PAR.K40_AtlasCopcoInputs[1].25;
//    P3_Srobovanie.STAV.K40_DosiahnutyMoment.2:= P3_Srobovanie.PAR.K40_AtlasCopcoInputs[1].26;
//    P3_Srobovanie.STAV.K40_DosiahnutyMoment.3:= P3_Srobovanie.PAR.K40_AtlasCopcoInputs[1].27;
//    P3_Srobovanie.STAV.K40_DosiahnutyMoment.4:= P3_Srobovanie.PAR.K40_AtlasCopcoInputs[1].28;
//    P3_Srobovanie.STAV.K40_DosiahnutyMoment.5:= P3_Srobovanie.PAR.K40_AtlasCopcoInputs[1].29;
//    P3_Srobovanie.STAV.K40_DosiahnutyMoment.6:= P3_Srobovanie.PAR.K40_AtlasCopcoInputs[1].30;
//    P3_Srobovanie.STAV.K40_DosiahnutyMoment.7:= P3_Srobovanie.PAR.K40_AtlasCopcoInputs[1].31;
//    P3_Srobovanie.STAV.K40_DosiahnutyMoment.8:= P3_Srobovanie.PAR.K40_AtlasCopcoInputs[1].16;
//    P3_Srobovanie.STAV.K40_DosiahnutyMoment.9:= P3_Srobovanie.PAR.K40_AtlasCopcoInputs[1].17;
//    P3_Srobovanie.STAV.K40_DosiahnutyMoment.10:= P3_Srobovanie.PAR.K40_AtlasCopcoInputs[1].18;
//    P3_Srobovanie.STAV.K40_DosiahnutyMoment.11:= P3_Srobovanie.PAR.K40_AtlasCopcoInputs[1].19;
//    P3_Srobovanie.STAV.K40_DosiahnutyMoment.12:= P3_Srobovanie.PAR.K40_AtlasCopcoInputs[1].20;
//    P3_Srobovanie.STAV.K40_DosiahnutyMoment.13:= P3_Srobovanie.PAR.K40_AtlasCopcoInputs[1].21;
//    P3_Srobovanie.STAV.K40_DosiahnutyMoment.14:= P3_Srobovanie.PAR.K40_AtlasCopcoInputs[1].22;
//    P3_Srobovanie.STAV.K40_DosiahnutyMoment.15:= P3_Srobovanie.PAR.K40_AtlasCopcoInputs[1].23;
//    P3_Srobovanie.STAV.K40_DosiahnutyMoment.16:= P3_Srobovanie.PAR.K40_AtlasCopcoInputs[1].8;
//    P3_Srobovanie.STAV.K40_DosiahnutyMoment.17:= P3_Srobovanie.PAR.K40_AtlasCopcoInputs[1].9;
//    P3_Srobovanie.STAV.K40_DosiahnutyMoment.18:= P3_Srobovanie.PAR.K40_AtlasCopcoInputs[1].10;
//    P3_Srobovanie.STAV.K40_DosiahnutyMoment.19:= P3_Srobovanie.PAR.K40_AtlasCopcoInputs[1].11;
//    P3_Srobovanie.STAV.K40_DosiahnutyMoment.20:= P3_Srobovanie.PAR.K40_AtlasCopcoInputs[1].12;
//    P3_Srobovanie.STAV.K40_DosiahnutyMoment.21:= P3_Srobovanie.PAR.K40_AtlasCopcoInputs[1].13;
//    P3_Srobovanie.STAV.K40_DosiahnutyMoment.22:= P3_Srobovanie.PAR.K40_AtlasCopcoInputs[1].14;
//    P3_Srobovanie.STAV.K40_DosiahnutyMoment.23:= P3_Srobovanie.PAR.K40_AtlasCopcoInputs[1].15;
//    P3_Srobovanie.STAV.K40_DosiahnutyMoment.24:= P3_Srobovanie.PAR.K40_AtlasCopcoInputs[1].0;
//    P3_Srobovanie.STAV.K40_DosiahnutyMoment.25:= P3_Srobovanie.PAR.K40_AtlasCopcoInputs[1].1;
//    P3_Srobovanie.STAV.K40_DosiahnutyMoment.26:= P3_Srobovanie.PAR.K40_AtlasCopcoInputs[1].2;
//    P3_Srobovanie.STAV.K40_DosiahnutyMoment.27:= P3_Srobovanie.PAR.K40_AtlasCopcoInputs[1].3;
//    P3_Srobovanie.STAV.K40_DosiahnutyMoment.28:= P3_Srobovanie.PAR.K40_AtlasCopcoInputs[1].4;
//    P3_Srobovanie.STAV.K40_DosiahnutyMoment.29:= P3_Srobovanie.PAR.K40_AtlasCopcoInputs[1].5;
//    P3_Srobovanie.STAV.K40_DosiahnutyMoment.30:= P3_Srobovanie.PAR.K40_AtlasCopcoInputs[1].6;
//    P3_Srobovanie.STAV.K40_DosiahnutyMoment.31:= P3_Srobovanie.PAR.K40_AtlasCopcoInputs[1].7;
//    K40_DosiahnutyMoment_REAL:= UDINT_TO_REAL(P3_Srobovanie.STAV.K40_DosiahnutyMoment);
//    IF K40_DosiahnutyMoment_REAL > 0 THEN
//        P3_Srobovanie.STAV.K40_DosiahnutyMoment_REAL:= (K40_DosiahnutyMoment_REAL*1.35)/65571;
//    ELSE
//        P3_Srobovanie.STAV.K40_DosiahnutyMoment_REAL:=0.0;
//    END_IF

    K40_PrevodMomentu.AtlasAktualnyMoment:=P3_Srobovanie.PAR.K40_AtlasCopcoInputs[1];
    P3_Srobovanie.STAV.K40_DosiahnutyMoment_REAL:=K40_PrevodMomentu.AktualnyMoment;

    (*P3_Srobovanie.STAV.K40_DosiahnutyMoment_REAL:= K40_DosiahnutyMoment_REAL/100;*)

    //Moment - Tolerancia MAX//
//    P3_Srobovanie.STAV.K40_Moment_ToleranciaMAX.0:= P3_Srobovanie.PAR.K40_AtlasCopcoInputs[3].24;
//    P3_Srobovanie.STAV.K40_Moment_ToleranciaMAX.1:= P3_Srobovanie.PAR.K40_AtlasCopcoInputs[3].25;
//    P3_Srobovanie.STAV.K40_Moment_ToleranciaMAX.2:= P3_Srobovanie.PAR.K40_AtlasCopcoInputs[3].26;
//    P3_Srobovanie.STAV.K40_Moment_ToleranciaMAX.3:= P3_Srobovanie.PAR.K40_AtlasCopcoInputs[3].27;
//    P3_Srobovanie.STAV.K40_Moment_ToleranciaMAX.4:= P3_Srobovanie.PAR.K40_AtlasCopcoInputs[3].28;
//    P3_Srobovanie.STAV.K40_Moment_ToleranciaMAX.5:= P3_Srobovanie.PAR.K40_AtlasCopcoInputs[3].29;
//    P3_Srobovanie.STAV.K40_Moment_ToleranciaMAX.6:= P3_Srobovanie.PAR.K40_AtlasCopcoInputs[3].30;
//    P3_Srobovanie.STAV.K40_Moment_ToleranciaMAX.7:= P3_Srobovanie.PAR.K40_AtlasCopcoInputs[3].31;
//    P3_Srobovanie.STAV.K40_Moment_ToleranciaMAX.8:= P3_Srobovanie.PAR.K40_AtlasCopcoInputs[3].16;
//    P3_Srobovanie.STAV.K40_Moment_ToleranciaMAX.9:= P3_Srobovanie.PAR.K40_AtlasCopcoInputs[3].17;
//    P3_Srobovanie.STAV.K40_Moment_ToleranciaMAX.10:= P3_Srobovanie.PAR.K40_AtlasCopcoInputs[3].18;
//    P3_Srobovanie.STAV.K40_Moment_ToleranciaMAX.11:= P3_Srobovanie.PAR.K40_AtlasCopcoInputs[3].19;
//    P3_Srobovanie.STAV.K40_Moment_ToleranciaMAX.12:= P3_Srobovanie.PAR.K40_AtlasCopcoInputs[3].20;
//    P3_Srobovanie.STAV.K40_Moment_ToleranciaMAX.13:= P3_Srobovanie.PAR.K40_AtlasCopcoInputs[3].21;
//    P3_Srobovanie.STAV.K40_Moment_ToleranciaMAX.14:= P3_Srobovanie.PAR.K40_AtlasCopcoInputs[3].22;
//    P3_Srobovanie.STAV.K40_Moment_ToleranciaMAX.15:= P3_Srobovanie.PAR.K40_AtlasCopcoInputs[3].23;
//    P3_Srobovanie.STAV.K40_Moment_ToleranciaMAX.16:= P3_Srobovanie.PAR.K40_AtlasCopcoInputs[3].8;
//    P3_Srobovanie.STAV.K40_Moment_ToleranciaMAX.17:= P3_Srobovanie.PAR.K40_AtlasCopcoInputs[3].9;
//    P3_Srobovanie.STAV.K40_Moment_ToleranciaMAX.18:= P3_Srobovanie.PAR.K40_AtlasCopcoInputs[3].10;
//    P3_Srobovanie.STAV.K40_Moment_ToleranciaMAX.19:= P3_Srobovanie.PAR.K40_AtlasCopcoInputs[3].11;
//    P3_Srobovanie.STAV.K40_Moment_ToleranciaMAX.20:= P3_Srobovanie.PAR.K40_AtlasCopcoInputs[3].12;
//    P3_Srobovanie.STAV.K40_Moment_ToleranciaMAX.21:= P3_Srobovanie.PAR.K40_AtlasCopcoInputs[3].13;
//    P3_Srobovanie.STAV.K40_Moment_ToleranciaMAX.22:= P3_Srobovanie.PAR.K40_AtlasCopcoInputs[3].14;
//    P3_Srobovanie.STAV.K40_Moment_ToleranciaMAX.23:= P3_Srobovanie.PAR.K40_AtlasCopcoInputs[3].15;
//    P3_Srobovanie.STAV.K40_Moment_ToleranciaMAX.24:= P3_Srobovanie.PAR.K40_AtlasCopcoInputs[3].0;
//    P3_Srobovanie.STAV.K40_Moment_ToleranciaMAX.25:= P3_Srobovanie.PAR.K40_AtlasCopcoInputs[3].1;
//    P3_Srobovanie.STAV.K40_Moment_ToleranciaMAX.26:= P3_Srobovanie.PAR.K40_AtlasCopcoInputs[3].2;
//    P3_Srobovanie.STAV.K40_Moment_ToleranciaMAX.27:= P3_Srobovanie.PAR.K40_AtlasCopcoInputs[3].3;
//    P3_Srobovanie.STAV.K40_Moment_ToleranciaMAX.28:= P3_Srobovanie.PAR.K40_AtlasCopcoInputs[3].4;
//    P3_Srobovanie.STAV.K40_Moment_ToleranciaMAX.29:= P3_Srobovanie.PAR.K40_AtlasCopcoInputs[3].5;
//    P3_Srobovanie.STAV.K40_Moment_ToleranciaMAX.30:= P3_Srobovanie.PAR.K40_AtlasCopcoInputs[3].6;
//    P3_Srobovanie.STAV.K40_Moment_ToleranciaMAX.31:= P3_Srobovanie.PAR.K40_AtlasCopcoInputs[3].7;
//    K40_Moment_ToleranciaMAX_REAL:= UDINT_TO_REAL(P3_Srobovanie.STAV.K40_Moment_ToleranciaMAX);
//    IF K40_Moment_ToleranciaMAX_REAL > 0 THEN
//       P3_Srobovanie.STAV.K40_Moment_ToleranciaMAX_REAL:= (K40_Moment_ToleranciaMAX_REAL*1.65)/65601;
//    ELSE
//        P3_Srobovanie.STAV.K40_Moment_ToleranciaMAX_REAL:= 0.0;
//    END_IF

    K40_PrevodMomentu.AtlasMaximalnaTolerancia:=P3_Srobovanie.PAR.K40_AtlasCopcoInputs[3];
    P3_Srobovanie.STAV.K40_Moment_ToleranciaMAX_REAL:=K40_PrevodMomentu.ToleranciaMAX;

    (*P3_Srobovanie.STAV.K40_Moment_ToleranciaMAX_REAL:= K40_Moment_ToleranciaMAX_REAL/100;*)

    //Moment - Tolerancia MIN//
//    P3_Srobovanie.STAV.K40_Moment_ToleranciaMIN.0:= P3_Srobovanie.PAR.K40_AtlasCopcoInputs[4].24;
//    P3_Srobovanie.STAV.K40_Moment_ToleranciaMIN.1:= P3_Srobovanie.PAR.K40_AtlasCopcoInputs[4].25;
//    P3_Srobovanie.STAV.K40_Moment_ToleranciaMIN.2:= P3_Srobovanie.PAR.K40_AtlasCopcoInputs[4].26;
//    P3_Srobovanie.STAV.K40_Moment_ToleranciaMIN.3:= P3_Srobovanie.PAR.K40_AtlasCopcoInputs[4].27;
//    P3_Srobovanie.STAV.K40_Moment_ToleranciaMIN.4:= P3_Srobovanie.PAR.K40_AtlasCopcoInputs[4].28;
//    P3_Srobovanie.STAV.K40_Moment_ToleranciaMIN.5:= P3_Srobovanie.PAR.K40_AtlasCopcoInputs[4].29;
//    P3_Srobovanie.STAV.K40_Moment_ToleranciaMIN.6:= P3_Srobovanie.PAR.K40_AtlasCopcoInputs[4].30;
//    P3_Srobovanie.STAV.K40_Moment_ToleranciaMIN.7:= P3_Srobovanie.PAR.K40_AtlasCopcoInputs[4].31;
//    P3_Srobovanie.STAV.K40_Moment_ToleranciaMIN.8:= P3_Srobovanie.PAR.K40_AtlasCopcoInputs[4].16;
//    P3_Srobovanie.STAV.K40_Moment_ToleranciaMIN.9:= P3_Srobovanie.PAR.K40_AtlasCopcoInputs[4].17;
//    P3_Srobovanie.STAV.K40_Moment_ToleranciaMIN.10:= P3_Srobovanie.PAR.K40_AtlasCopcoInputs[4].18;
//    P3_Srobovanie.STAV.K40_Moment_ToleranciaMIN.11:= P3_Srobovanie.PAR.K40_AtlasCopcoInputs[4].19;
//    P3_Srobovanie.STAV.K40_Moment_ToleranciaMIN.12:= P3_Srobovanie.PAR.K40_AtlasCopcoInputs[4].20;
//    P3_Srobovanie.STAV.K40_Moment_ToleranciaMIN.13:= P3_Srobovanie.PAR.K40_AtlasCopcoInputs[4].21;
//    P3_Srobovanie.STAV.K40_Moment_ToleranciaMIN.14:= P3_Srobovanie.PAR.K40_AtlasCopcoInputs[4].22;
//    P3_Srobovanie.STAV.K40_Moment_ToleranciaMIN.15:= P3_Srobovanie.PAR.K40_AtlasCopcoInputs[4].23;
//    P3_Srobovanie.STAV.K40_Moment_ToleranciaMIN.16:= P3_Srobovanie.PAR.K40_AtlasCopcoInputs[4].8;
//    P3_Srobovanie.STAV.K40_Moment_ToleranciaMIN.17:= P3_Srobovanie.PAR.K40_AtlasCopcoInputs[4].9;
//    P3_Srobovanie.STAV.K40_Moment_ToleranciaMIN.18:= P3_Srobovanie.PAR.K40_AtlasCopcoInputs[4].10;
//    P3_Srobovanie.STAV.K40_Moment_ToleranciaMIN.19:= P3_Srobovanie.PAR.K40_AtlasCopcoInputs[4].11;
//    P3_Srobovanie.STAV.K40_Moment_ToleranciaMIN.20:= P3_Srobovanie.PAR.K40_AtlasCopcoInputs[4].12;
//    P3_Srobovanie.STAV.K40_Moment_ToleranciaMIN.21:= P3_Srobovanie.PAR.K40_AtlasCopcoInputs[4].13;
//    P3_Srobovanie.STAV.K40_Moment_ToleranciaMIN.22:= P3_Srobovanie.PAR.K40_AtlasCopcoInputs[4].14;
//    P3_Srobovanie.STAV.K40_Moment_ToleranciaMIN.23:= P3_Srobovanie.PAR.K40_AtlasCopcoInputs[4].15;
//    P3_Srobovanie.STAV.K40_Moment_ToleranciaMIN.24:= P3_Srobovanie.PAR.K40_AtlasCopcoInputs[4].0;
//    P3_Srobovanie.STAV.K40_Moment_ToleranciaMIN.25:= P3_Srobovanie.PAR.K40_AtlasCopcoInputs[4].1;
//    P3_Srobovanie.STAV.K40_Moment_ToleranciaMIN.26:= P3_Srobovanie.PAR.K40_AtlasCopcoInputs[4].2;
//    P3_Srobovanie.STAV.K40_Moment_ToleranciaMIN.27:= P3_Srobovanie.PAR.K40_AtlasCopcoInputs[4].3;
//    P3_Srobovanie.STAV.K40_Moment_ToleranciaMIN.28:= P3_Srobovanie.PAR.K40_AtlasCopcoInputs[4].4;
//    P3_Srobovanie.STAV.K40_Moment_ToleranciaMIN.29:= P3_Srobovanie.PAR.K40_AtlasCopcoInputs[4].5;
//    P3_Srobovanie.STAV.K40_Moment_ToleranciaMIN.30:= P3_Srobovanie.PAR.K40_AtlasCopcoInputs[4].6;
//    P3_Srobovanie.STAV.K40_Moment_ToleranciaMIN.31:= P3_Srobovanie.PAR.K40_AtlasCopcoInputs[4].7;
//    K40_Moment_ToleranciaMIN_REAL:= UDINT_TO_REAL(P3_Srobovanie.STAV.K40_Moment_ToleranciaMIN);
//    IF K40_Moment_ToleranciaMIN_REAL > 0 THEN
//      P3_Srobovanie.STAV.K40_Moment_ToleranciaMIN_REAL:= (K40_Moment_ToleranciaMIN_REAL*1.35)/65571;
//    ELSE
//        P3_Srobovanie.STAV.K40_Moment_ToleranciaMIN_REAL:=0.0;
//    END_IF

    K40_PrevodMomentu.AtlasMinimalnaTolerancia:=P3_Srobovanie.PAR.K40_AtlasCopcoInputs[4];
    P3_Srobovanie.STAV.K40_Moment_ToleranciaMIN_REAL:=K40_PrevodMomentu.ToleranciaMIN;

    (*P3_Srobovanie.STAV.K40_Moment_ToleranciaMIN_REAL:= K40_Moment_ToleranciaMIN_REAL /100;*)

    //Dosiahnutý úhol//
    P3_Srobovanie.STAV.K40_DosiahnutyUhol.0:= P3_Srobovanie.PAR.K40_AtlasCopcoInputs[0].24;
    P3_Srobovanie.STAV.K40_DosiahnutyUhol.1:= P3_Srobovanie.PAR.K40_AtlasCopcoInputs[0].25;
    P3_Srobovanie.STAV.K40_DosiahnutyUhol.2:= P3_Srobovanie.PAR.K40_AtlasCopcoInputs[0].26;
    P3_Srobovanie.STAV.K40_DosiahnutyUhol.3:= P3_Srobovanie.PAR.K40_AtlasCopcoInputs[0].27;
    P3_Srobovanie.STAV.K40_DosiahnutyUhol.4:= P3_Srobovanie.PAR.K40_AtlasCopcoInputs[0].28;
    P3_Srobovanie.STAV.K40_DosiahnutyUhol.5:= P3_Srobovanie.PAR.K40_AtlasCopcoInputs[0].29;
    P3_Srobovanie.STAV.K40_DosiahnutyUhol.6:= P3_Srobovanie.PAR.K40_AtlasCopcoInputs[0].30;
    P3_Srobovanie.STAV.K40_DosiahnutyUhol.7:= P3_Srobovanie.PAR.K40_AtlasCopcoInputs[0].31;
    P3_Srobovanie.STAV.K40_DosiahnutyUhol.8:= P3_Srobovanie.PAR.K40_AtlasCopcoInputs[0].16;
    P3_Srobovanie.STAV.K40_DosiahnutyUhol.9:= P3_Srobovanie.PAR.K40_AtlasCopcoInputs[0].17;
    P3_Srobovanie.STAV.K40_DosiahnutyUhol.10:= P3_Srobovanie.PAR.K40_AtlasCopcoInputs[0].18;
    P3_Srobovanie.STAV.K40_DosiahnutyUhol.11:= P3_Srobovanie.PAR.K40_AtlasCopcoInputs[0].19;
    P3_Srobovanie.STAV.K40_DosiahnutyUhol.12:= P3_Srobovanie.PAR.K40_AtlasCopcoInputs[0].20;
    P3_Srobovanie.STAV.K40_DosiahnutyUhol.13:= P3_Srobovanie.PAR.K40_AtlasCopcoInputs[0].21;
    P3_Srobovanie.STAV.K40_DosiahnutyUhol.14:= P3_Srobovanie.PAR.K40_AtlasCopcoInputs[0].22;
    P3_Srobovanie.STAV.K40_DosiahnutyUhol.15:= P3_Srobovanie.PAR.K40_AtlasCopcoInputs[0].23;

    //Uhol - Tolerancia MAX//
    P3_Srobovanie.STAV.K40_Uhol_ToleranciaMAX.0:= P3_Srobovanie.PAR.K40_AtlasCopcoInputs[2].8;
    P3_Srobovanie.STAV.K40_Uhol_ToleranciaMAX.1:= P3_Srobovanie.PAR.K40_AtlasCopcoInputs[2].9;
    P3_Srobovanie.STAV.K40_Uhol_ToleranciaMAX.2:= P3_Srobovanie.PAR.K40_AtlasCopcoInputs[2].10;
    P3_Srobovanie.STAV.K40_Uhol_ToleranciaMAX.3:= P3_Srobovanie.PAR.K40_AtlasCopcoInputs[2].11;
    P3_Srobovanie.STAV.K40_Uhol_ToleranciaMAX.4:= P3_Srobovanie.PAR.K40_AtlasCopcoInputs[2].12;
    P3_Srobovanie.STAV.K40_Uhol_ToleranciaMAX.5:= P3_Srobovanie.PAR.K40_AtlasCopcoInputs[2].13;
    P3_Srobovanie.STAV.K40_Uhol_ToleranciaMAX.6:= P3_Srobovanie.PAR.K40_AtlasCopcoInputs[2].14;
    P3_Srobovanie.STAV.K40_Uhol_ToleranciaMAX.7:= P3_Srobovanie.PAR.K40_AtlasCopcoInputs[2].15;
    P3_Srobovanie.STAV.K40_Uhol_ToleranciaMAX.8:= P3_Srobovanie.PAR.K40_AtlasCopcoInputs[2].0;
    P3_Srobovanie.STAV.K40_Uhol_ToleranciaMAX.9:= P3_Srobovanie.PAR.K40_AtlasCopcoInputs[2].1;
    P3_Srobovanie.STAV.K40_Uhol_ToleranciaMAX.10:= P3_Srobovanie.PAR.K40_AtlasCopcoInputs[2].2;
    P3_Srobovanie.STAV.K40_Uhol_ToleranciaMAX.11:= P3_Srobovanie.PAR.K40_AtlasCopcoInputs[2].3;
    P3_Srobovanie.STAV.K40_Uhol_ToleranciaMAX.12:= P3_Srobovanie.PAR.K40_AtlasCopcoInputs[2].4;
    P3_Srobovanie.STAV.K40_Uhol_ToleranciaMAX.13:= P3_Srobovanie.PAR.K40_AtlasCopcoInputs[2].5;
    P3_Srobovanie.STAV.K40_Uhol_ToleranciaMAX.14:= P3_Srobovanie.PAR.K40_AtlasCopcoInputs[2].6;
    P3_Srobovanie.STAV.K40_Uhol_ToleranciaMAX.15:= P3_Srobovanie.PAR.K40_AtlasCopcoInputs[2].7;

    //Uhol - Tolerancia MIN//
    P3_Srobovanie.STAV.K40_Uhol_ToleranciaMIN.0:= P3_Srobovanie.PAR.K40_AtlasCopcoInputs[2].24;
    P3_Srobovanie.STAV.K40_Uhol_ToleranciaMIN.1:= P3_Srobovanie.PAR.K40_AtlasCopcoInputs[2].25;
    P3_Srobovanie.STAV.K40_Uhol_ToleranciaMIN.2:= P3_Srobovanie.PAR.K40_AtlasCopcoInputs[2].26;
    P3_Srobovanie.STAV.K40_Uhol_ToleranciaMIN.3:= P3_Srobovanie.PAR.K40_AtlasCopcoInputs[2].27;
    P3_Srobovanie.STAV.K40_Uhol_ToleranciaMIN.4:= P3_Srobovanie.PAR.K40_AtlasCopcoInputs[2].28;
    P3_Srobovanie.STAV.K40_Uhol_ToleranciaMIN.5:= P3_Srobovanie.PAR.K40_AtlasCopcoInputs[2].29;
    P3_Srobovanie.STAV.K40_Uhol_ToleranciaMIN.6:= P3_Srobovanie.PAR.K40_AtlasCopcoInputs[2].30;
    P3_Srobovanie.STAV.K40_Uhol_ToleranciaMIN.7:= P3_Srobovanie.PAR.K40_AtlasCopcoInputs[2].31;
    P3_Srobovanie.STAV.K40_Uhol_ToleranciaMIN.8:= P3_Srobovanie.PAR.K40_AtlasCopcoInputs[2].16;
    P3_Srobovanie.STAV.K40_Uhol_ToleranciaMIN.9:= P3_Srobovanie.PAR.K40_AtlasCopcoInputs[2].17;
    P3_Srobovanie.STAV.K40_Uhol_ToleranciaMIN.10:= P3_Srobovanie.PAR.K40_AtlasCopcoInputs[2].18;
    P3_Srobovanie.STAV.K40_Uhol_ToleranciaMIN.11:= P3_Srobovanie.PAR.K40_AtlasCopcoInputs[2].19;
    P3_Srobovanie.STAV.K40_Uhol_ToleranciaMIN.12:= P3_Srobovanie.PAR.K40_AtlasCopcoInputs[2].20;
    P3_Srobovanie.STAV.K40_Uhol_ToleranciaMIN.13:= P3_Srobovanie.PAR.K40_AtlasCopcoInputs[2].21;
    P3_Srobovanie.STAV.K40_Uhol_ToleranciaMIN.14:= P3_Srobovanie.PAR.K40_AtlasCopcoInputs[2].22;
    P3_Srobovanie.STAV.K40_Uhol_ToleranciaMIN.15:= P3_Srobovanie.PAR.K40_AtlasCopcoInputs[2].23;

END_ACTION
```

#### OvlZdvihuHV_Testu.st
```iecst
ACTION OvlZdvihuHV_Testu:

	//Volanie funkcie SequenceControl//
	SequenceControl(SC:= SC_OvlZdvihuHV_Testu);

	CASE SC_OvlZdvihuHV_Testu.Step OF

		0:
			SC_OvlZdvihuHV_Testu.StepName:= '0 - Nulovanie';
			HV_Test_VYSUN:= FALSE;
			HV_Test_ZASUN:= FALSE;
//			P3_Srobovanie.OUT.HVTest_VYSUN_YV150:= FALSE;
//			P3_Srobovanie.OUT.HVTest_ZASUN_YV149:= FALSE;

			IF SC_P3_Srobovanie.Step <> 0 THEN
				SC_OvlZdvihuHV_Testu.ResetStep:= TRUE;
				SC_OvlZdvihuHV_Testu.Step:= 1;
			END_IF

		1:
			SC_OvlZdvihuHV_Testu.StepName:= '1 - Rozhodnutie o cinnosti';
			IF HV_Test_VYSUN THEN
				SC_OvlZdvihuHV_Testu.Step:= 10;
			ELSIF HV_Test_ZASUN THEN
				SC_OvlZdvihuHV_Testu.Step:= 20;
			END_IF

		10:
			SC_OvlZdvihuHV_Testu.StepName:= '10 - Vysunutie HV testu';
			SC_OvlZdvihuHV_Testu.IdleTime.PT:= T#3s;
			SC_OvlZdvihuHV_Testu.AlarmTime.PT:= T#10s;

			IF P3_Srobovanie.Automat THEN
				SC_OvlZdvihuHV_Testu.AlarmTime.IN:= TRUE;
			ELSE
				SC_OvlZdvihuHV_Testu.IdleTime.IN:= TRUE;
			END_IF

			IF NOT SC_OvlZdvihuHV_Testu.Switch1 THEN
				P3_Srobovanie.OUT.HVTest_ZASUN_YV149:= FALSE;
				P3_Srobovanie.OUT.HVTest_VYSUN_YV150:= TRUE;
				SC_OvlZdvihuHV_Testu.Switch1:= TRUE;
			END_IF

			IF P3_Srobovanie.IN.HVTest_VYSUNUTY_MS50 OR SC_OvlZdvihuHV_Testu.IdleTime.Q THEN
				SC_OvlZdvihuHV_Testu.ResetStep:= TRUE;
				SC_OvlZdvihuHV_Testu.Step:= 0;
			ELSIF SC_OvlZdvihuHV_Testu.AlarmTime.Q THEN
				P34_Alarmy[318]:= TRUE;
				P3_PoruchaST1:= TRUE;
			END_IF

		20:
			SC_OvlZdvihuHV_Testu.StepName:= '20 - Zasunutie HV testu';
			SC_OvlZdvihuHV_Testu.IdleTime.PT:= T#3s;
			SC_OvlZdvihuHV_Testu.AlarmTime.PT:= T#10s;

			IF P3_Srobovanie.Automat THEN
				SC_OvlZdvihuHV_Testu.AlarmTime.IN:= TRUE;
			ELSE
				SC_OvlZdvihuHV_Testu.IdleTime.IN:= TRUE;
			END_IF

			IF NOT SC_OvlZdvihuHV_Testu.Switch1 THEN
				P3_Srobovanie.OUT.HVTest_VYSUN_YV150:= FALSE;
				P3_Srobovanie.OUT.HVTest_ZASUN_YV149:= TRUE;
				SC_OvlZdvihuHV_Testu.Switch1:= TRUE;
			END_IF

			IF P3_Srobovanie.IN.HVTest_ZASUNUTY_MS51 OR SC_OvlZdvihuHV_Testu.IdleTime.Q THEN
				SC_OvlZdvihuHV_Testu.ResetStep:= TRUE;
				SC_OvlZdvihuHV_Testu.Step:= 0;
			ELSIF SC_OvlZdvihuHV_Testu.AlarmTime.Q THEN
				P34_Alarmy[319]:= TRUE;
				P3_PoruchaST1:= TRUE;
			END_IF

	END_CASE

END_ACTION
```

#### OvlKontaktovHV_Testu.st
```iecst
ACTION OvlKontaktovHV_Testu:

	//Volanie funkcie SequenceControl//
	SequenceControl(SC:= SC_OvlKontaktovHV_Testu);

	CASE SC_OvlKontaktovHV_Testu.Step OF

		0:
			SC_OvlKontaktovHV_Testu.StepName:= '0 - Nulovanie';
			Kontakty_VYSUN:= FALSE;
			Kontakty_ZASUN:= FALSE;
//			P3_Srobovanie.OUT.HVTest_Kontakty_VYSUN_YV154:= FALSE;
//			P3_Srobovanie.OUT.HVTest_Kontakty_ZASUN_YV153:= FALSE;

			IF SC_P3_Srobovanie.Step <> 0 THEN
				SC_OvlKontaktovHV_Testu.ResetStep:= TRUE;
				SC_OvlKontaktovHV_Testu.Step:= 1;
			END_IF

		1:
			SC_OvlKontaktovHV_Testu.StepName:= '1 - Rozhodnutie o cinnosti';
			IF Kontakty_VYSUN THEN
				SC_OvlKontaktovHV_Testu.Step:= 10;
			ELSIF Kontakty_ZASUN THEN
				SC_OvlKontaktovHV_Testu.Step:= 20;
			END_IF

		10:
			SC_OvlKontaktovHV_Testu.StepName:= '10 - Vysunutie kontaktov HV testu';
			SC_OvlKontaktovHV_Testu.IdleTime.PT:= T#3s;
			SC_OvlKontaktovHV_Testu.AlarmTime.PT:= T#20s;

			IF P3_Srobovanie.Automat THEN
				SC_OvlKontaktovHV_Testu.AlarmTime.IN:= TRUE;
			ELSE
				SC_OvlKontaktovHV_Testu.IdleTime.IN:= TRUE;
			END_IF

			IF NOT SC_OvlKontaktovHV_Testu.Switch1 THEN
				P3_Srobovanie.OUT.HVTest_Kontakty_ZASUN_YV153:= FALSE;
				P3_Srobovanie.OUT.HVTest_Kontakty_VYSUN_YV154:= TRUE;
				SC_OvlKontaktovHV_Testu.Switch1:= TRUE;
			END_IF

			IF P3_Srobovanie.IN.HVTest_Kontakty_VYSUNUTE_MS45 OR SC_OvlKontaktovHV_Testu.IdleTime.Q THEN
				SC_OvlKontaktovHV_Testu.ResetStep:= TRUE;
				SC_OvlKontaktovHV_Testu.Step:= 0;
			ELSIF SC_OvlKontaktovHV_Testu.AlarmTime.Q THEN
				P34_Alarmy[316]:= TRUE;
				P3_PoruchaST1:= TRUE;
			END_IF

		20:
			SC_OvlKontaktovHV_Testu.StepName:= '20 - Zasunutie kontaktov HV testu';
			SC_OvlKontaktovHV_Testu.IdleTime.PT:= T#3s;
			SC_OvlKontaktovHV_Testu.AlarmTime.PT:= T#20s;

			IF P3_Srobovanie.Automat THEN
				SC_OvlKontaktovHV_Testu.AlarmTime.IN:= TRUE;
			ELSE
				SC_OvlKontaktovHV_Testu.IdleTime.IN:= TRUE;
			END_IF

			IF NOT SC_OvlKontaktovHV_Testu.Switch1 THEN
				P3_Srobovanie.OUT.HVTest_Kontakty_VYSUN_YV154:= FALSE;
				P3_Srobovanie.OUT.HVTest_Kontakty_ZASUN_YV153:= TRUE;
				SC_OvlKontaktovHV_Testu.Switch1:= TRUE;
			END_IF

			IF P3_Srobovanie.IN.HVTest_Kontakty_ZASUNUTE_MS44 OR SC_OvlKontaktovHV_Testu.IdleTime.Q THEN
				SC_OvlKontaktovHV_Testu.ResetStep:= TRUE;
				SC_OvlKontaktovHV_Testu.Step:= 0;
			ELSIF SC_OvlKontaktovHV_Testu.AlarmTime.Q THEN
				P34_Alarmy[317]:= TRUE;
				P3_PoruchaST1:= TRUE;
			END_IF

	END_CASE

END_ACTION
```

#### OvlTestera.st
```iecst
ACTION OvlTestera:

	//Parametre komunikácie//
    memcpy(ADR(SKTcpClientTester_0.Params.IPaddrServ),ADR('192.168.122.251'),SIZEOF('192.168.122.251'));
    SKTcpClientTester_0.Params.IPportClient := 1031;
    SKTcpClientTester_0.Params.IPportServ := 1030;
    SKTcpClientTester_0.Params.RecvTimeout := 10000;
    strcpy(ADR(SKTcpClientTester_0.Params.Packet.data),ADR(dataStr));
    SKTcpClientTester_0();

    Cas_HVTester.PT:= T#1M;
    Cas_HVTester();

    //Volanie funkcie SequenceControl//
    SequenceControl(SC:= SC_OvlTesteraHV);

    CASE SC_OvlTesteraHV.Step OF

        0:
            SC_OvlTesteraHV.StepName:= '0 - Nulovanie';
            SKTcpClientTester_0.Enable:= TRUE;
            SKTcpClientTester_0.Cmd.Send:= FALSE;
            HV_Test_UKONCENY:= FALSE;
            PocetDopytovNaTester:= 0;
            SC_OvlTesteraHV.ResetStep:= TRUE;
            SC_OvlTesteraHV.Step:= 1;

        1:
            SC_OvlTesteraHV.StepName:= '1 - Cakam na spustenie testera';
            IF HV_Test_START THEN
                P3_Srobovanie.STAV.Vysledok_HV_Testu:= '';
                Cas_HVTester.IN:= TRUE;
                NameranyCas_InitTestera:= 0;
                NameranyCas_PoslanieQRkodu:= 0;
                NameranyCas_CelkovyCasTestovania:= 0;
                SC_OvlTesteraHV.Step:= 10;
            END_IF

        10:
            SC_OvlTesteraHV.StepName:= '10 - Dopyt na stav testera - typ 0';
            SC_OvlTesteraHV.IdleTime.PT:= T#300ms;
            SC_OvlTesteraHV.AlarmTime.PT:= T#5s;
            SC_OvlTesteraHV.IdleTime.IN:= TRUE;
            SC_OvlTesteraHV.AlarmTime.IN:= TRUE;

            SKTcpClientTester_0.Params.Packet.type:= 0;
            SKTcpClientTester_0.Params.Packet.workplace:= 46;
            SKTcpClientTester_0.Params.Packet.id:= 1;
            SKTcpClientTester_0.Cmd.Send:= TRUE;

            IF SKTcpClientTester_0.Cmd.Send AND NOT SKTcpClientTester_0.Status.staReceived AND NOT SKTcpClientTester_0.Status.staError THEN
                SC_OvlTesteraHV.ResetStep:= TRUE;
                SC_OvlTesteraHV.Step:= 13;
            ELSIF SC_OvlTesteraHV.AlarmTime.Q AND (SKTcpClientTester_0.Status.staReceived OR SKTcpClientTester_0.Status.staError) THEN
                PocetDopytovNaTester:= PocetDopytovNaTester + 1;
                SC_OvlTesteraHV.ResetStep:= TRUE;
                SC_OvlTesteraHV.Step:= 12;
            END_IF

        12:
            SC_OvlTesteraHV.StepName:= '12 - Dopyt na stav testera - cakam na opatovny dopyt na tester';
            SC_OvlTesteraHV.IdleTime.PT:= T#300ms;
            SC_OvlTesteraHV.AlarmTime.PT:= T#5s;
            SC_OvlTesteraHV.IdleTime.IN:= TRUE;
            SKTcpClientTester_0.Cmd.Send:= FALSE;

            IF PocetDopytovNaTester < 3 THEN
                IF SC_OvlTesteraHV.IdleTime.Q THEN
                    SC_OvlTesteraHV.ResetStep:= TRUE;
                    SC_OvlTesteraHV.Step:= 10;
                END_IF
            ELSE
                P3_Srobovanie.STAV.Vysledok_HV_Testu:= 'NG';
                HV_Test_UKONCENY:= TRUE;
                SC_OvlTesteraHV.ResetStep:= TRUE;
                SC_OvlTesteraHV.Step:= 100;
            END_IF

        13:
            SC_OvlTesteraHV.StepName:= '13 - Odpoved na stav testera - typ 0';
            SC_OvlTesteraHV.IdleTime.PT:= T#500ms;
            SC_OvlTesteraHV.AlarmTime.PT:= T#10s;
            SC_OvlTesteraHV.IdleTime.IN:= TRUE;

            IF SKTcpClientTester_0.Status.staReceived AND SKTcpClientTester_0.Status.DataRecv[2]= 0 AND SKTcpClientTester_0.Status.DataRecv[5]= 2 THEN
                SKTcpClientTester_0.Cmd.Send:= FALSE;
                NameranyCas_InitTestera:= Cas_HVTester.ET;
                SC_OvlTesteraHV.ResetStep:= TRUE;
                SC_OvlTesteraHV.Step:= 15;
            ELSIF SKTcpClientTester_0.Status.staReceived AND SKTcpClientTester_0.Status.DataRecv[2]= 0 AND SKTcpClientTester_0.Status.DataRecv[5]= 1 THEN
                SKTcpClientTester_0.Cmd.Send:= FALSE;
                IF SC_OvlTesteraHV.IdleTime.Q THEN
                    SC_OvlTesteraHV.ResetStep:= TRUE;
                    SC_OvlTesteraHV.Step:= 10;
                END_IF
            ELSIF SKTcpClientTester_0.Status.staReceived AND SKTcpClientTester_0.Status.DataRecv[2]= 0 AND SKTcpClientTester_0.Status.DataRecv[5]= 0 THEN
                SKTcpClientTester_0.Cmd.Send:= FALSE;
                IF SC_OvlTesteraHV.IdleTime.Q THEN
                    SC_OvlTesteraHV.ResetStep:= TRUE;
                    SC_OvlTesteraHV.Step:= 10;
                END_IF
            ELSIF SKTcpClientTester_0.Status.staError THEN
                SKTcpClientTester_0.Cmd.Send:= FALSE;
                P3_Srobovanie.STAV.Vysledok_HV_Testu:= 'NG';
                HV_Test_UKONCENY:= TRUE;
                SC_OvlTesteraHV.ResetStep:= TRUE;
                SC_OvlTesteraHV.Step:= 100;
            END_IF

        15:
            SC_OvlTesteraHV.StepName:= '15 - Poslanie QR kodu Power CP - typ 1';
            SC_OvlTesteraHV.IdleTime.PT:= T#300ms;
            SC_OvlTesteraHV.AlarmTime.PT:= T#10s;
            SC_OvlTesteraHV.IdleTime.IN:= TRUE;

            SKTcpClientTester_0.Params.Packet.type:= 1;
            SKTcpClientTester_0.Params.Packet.workplace:= 46;
            SKTcpClientTester_0.Params.Packet.id:= 1;
            dataStr:= Paletka[i].PAR.QRkodPowerCP;
            SKTcpClientTester_0.Cmd.Send:= TRUE;

            IF SKTcpClientTester_0.Cmd.Send AND NOT SKTcpClientTester_0.Status.staReceived AND NOT SKTcpClientTester_0.Status.staError THEN
                SC_OvlTesteraHV.ResetStep:= TRUE;
                SC_OvlTesteraHV.Step:= 18;
            END_IF

        18:
            SC_OvlTesteraHV.StepName:= '18 - Odpoved na poslanie QR kodu - typ 1';
            SC_OvlTesteraHV.IdleTime.PT:= T#300ms;
            SC_OvlTesteraHV.AlarmTime.PT:= T#10s;
            SC_OvlTesteraHV.IdleTime.IN:= TRUE;

            IF SKTcpClientTester_0.Status.staReceived AND SKTcpClientTester_0.Status.DataRecv[2]= 1 AND SKTcpClientTester_0.Status.DataRecv[5]= 0 THEN
                SKTcpClientTester_0.Cmd.Send:= FALSE;
                NameranyCas_PoslanieQRkodu:= Cas_HVTester.ET;
                SC_OvlTesteraHV.ResetStep:= TRUE;
                SC_OvlTesteraHV.Step:= 20;
            ELSIF SKTcpClientTester_0.Status.staReceived AND SKTcpClientTester_0.Status.DataRecv[2]= 1 AND SKTcpClientTester_0.Status.DataRecv[5]= 2 THEN
                SKTcpClientTester_0.Cmd.Send:= FALSE;
                IF SC_OvlTesteraHV.IdleTime.Q THEN
                    SC_OvlTesteraHV.ResetStep:= TRUE;
                    SC_OvlTesteraHV.Step:= 15;
                END_IF
            ELSIF SKTcpClientTester_0.Status.staReceived AND SKTcpClientTester_0.Status.DataRecv[2]= 1 AND SKTcpClientTester_0.Status.DataRecv[5]= 1 THEN
                SKTcpClientTester_0.Cmd.Send:= FALSE;
                P3_Srobovanie.STAV.Vysledok_HV_Testu:= 'NG';
                HV_Test_UKONCENY:= TRUE;
                SC_OvlTesteraHV.ResetStep:= TRUE;
                SC_OvlTesteraHV.Step:= 100;
            ELSIF SKTcpClientTester_0.Status.staError THEN
                SKTcpClientTester_0.Cmd.Send:= FALSE;
                P3_Srobovanie.STAV.Vysledok_HV_Testu:= 'NG';
                HV_Test_UKONCENY:= TRUE;
                SC_OvlTesteraHV.ResetStep:= TRUE;
                SC_OvlTesteraHV.Step:= 100;
            END_IF

        20:
            SC_OvlTesteraHV.StepName:= '20 - Dopyt na stav testera - typ 0';
            SC_OvlTesteraHV.IdleTime.PT:= T#300ms;
            SC_OvlTesteraHV.AlarmTime.PT:= T#10s;
            SC_OvlTesteraHV.IdleTime.IN:= TRUE;

            SKTcpClientTester_0.Params.Packet.type:= 0;
            SKTcpClientTester_0.Params.Packet.workplace:= 46;
            SKTcpClientTester_0.Params.Packet.id:= 1;
            SKTcpClientTester_0.Cmd.Send:= TRUE;

            IF SKTcpClientTester_0.Cmd.Send AND NOT SKTcpClientTester_0.Status.staReceived AND NOT SKTcpClientTester_0.Status.staError THEN
                SC_OvlTesteraHV.ResetStep:= TRUE;
                SC_OvlTesteraHV.Step:= 23;
            END_IF

        23:
            SC_OvlTesteraHV.StepName:= '23 - Odpoved na stav testera - typ 0';
            SC_OvlTesteraHV.IdleTime.PT:= T#300ms;
            SC_OvlTesteraHV.AlarmTime.PT:= T#10s;
            SC_OvlTesteraHV.IdleTime.IN:= TRUE;

            IF SKTcpClientTester_0.Status.staReceived AND SKTcpClientTester_0.Status.DataRecv[2]= 0 AND SKTcpClientTester_0.Status.DataRecv[5]= 3 THEN
                SKTcpClientTester_0.Cmd.Send:= FALSE;
                IF SC_OvlTesteraHV.IdleTime.Q THEN
                    SC_OvlTesteraHV.ResetStep:= TRUE;
                    SC_OvlTesteraHV.Step:= 20;
                END_IF
            ELSIF SKTcpClientTester_0.Status.staReceived AND SKTcpClientTester_0.Status.DataRecv[2]= 0 AND SKTcpClientTester_0.Status.DataRecv[5]= 4 THEN
                SKTcpClientTester_0.Cmd.Send:= FALSE;
                SC_OvlTesteraHV.ResetStep:= TRUE;
                SC_OvlTesteraHV.Step:= 25;
            ELSIF SKTcpClientTester_0.Status.staReceived AND SKTcpClientTester_0.Status.DataRecv[2]= 0 AND SKTcpClientTester_0.Status.DataRecv[5]= 0 THEN
                SKTcpClientTester_0.Cmd.Send:= FALSE;
                P3_Srobovanie.STAV.Vysledok_HV_Testu:= 'NG';
                HV_Test_UKONCENY:= TRUE;
                SC_OvlTesteraHV.ResetStep:= TRUE;
                SC_OvlTesteraHV.Step:= 100;
            ELSIF SKTcpClientTester_0.Status.staError THEN
                SKTcpClientTester_0.Cmd.Send:= FALSE;
                P3_Srobovanie.STAV.Vysledok_HV_Testu:= 'NG';
                HV_Test_UKONCENY:= TRUE;
                SC_OvlTesteraHV.ResetStep:= TRUE;
                SC_OvlTesteraHV.Step:= 100;
            END_IF

        25:
            SC_OvlTesteraHV.StepName:= '25 - Dopyt na vysledok testu - typ 2';
            SC_OvlTesteraHV.IdleTime.PT:= T#300ms;
            SC_OvlTesteraHV.AlarmTime.PT:= T#10s;
            SC_OvlTesteraHV.IdleTime.IN:= TRUE;

            SKTcpClientTester_0.Params.Packet.type:= 2;
            SKTcpClientTester_0.Params.Packet.workplace:= 46;
            SKTcpClientTester_0.Params.Packet.id:= 1;
            SKTcpClientTester_0.Cmd.Send:= TRUE;

            IF SKTcpClientTester_0.Cmd.Send AND NOT SKTcpClientTester_0.Status.staReceived AND NOT SKTcpClientTester_0.Status.staError THEN
                SC_OvlTesteraHV.ResetStep:= TRUE;
                SC_OvlTesteraHV.Step:= 28;
            END_IF

        28:
            SC_OvlTesteraHV.StepName:= '28 - Odpoved na vysledok testu - typ 2';
            SC_OvlTesteraHV.IdleTime.PT:= T#300ms;
            SC_OvlTesteraHV.AlarmTime.PT:= T#10s;
            SC_OvlTesteraHV.IdleTime.IN:= TRUE;

            IF SKTcpClientTester_0.Status.staReceived AND SKTcpClientTester_0.Status.DataRecv[2]= 2 AND SKTcpClientTester_0.Status.DataRecv[5]= 1 THEN
                SKTcpClientTester_0.Cmd.Send:= FALSE;
                P3_Srobovanie.STAV.Vysledok_HV_Testu:= 'OK';
                SC_OvlTesteraHV.ResetStep:= TRUE;
                SC_OvlTesteraHV.Step:= 30;
            ELSIF SKTcpClientTester_0.Status.staReceived AND SKTcpClientTester_0.Status.DataRecv[2]= 2 AND SKTcpClientTester_0.Status.DataRecv[5]= 2 THEN
                SKTcpClientTester_0.Cmd.Send:= FALSE;
                P3_Srobovanie.STAV.Vysledok_HV_Testu:= 'NG';
                SC_OvlTesteraHV.ResetStep:= TRUE;
                SC_OvlTesteraHV.Step:= 30;
            ELSIF SKTcpClientTester_0.Status.staReceived AND SKTcpClientTester_0.Status.DataRecv[2]= 2 AND SKTcpClientTester_0.Status.DataRecv[5]= 0 THEN
                SKTcpClientTester_0.Cmd.Send:= FALSE;
                IF SC_OvlTesteraHV.IdleTime.Q THEN
                    SC_OvlTesteraHV.ResetStep:= TRUE;
                    SC_OvlTesteraHV.Step:= 25;
                END_IF
            ELSIF SKTcpClientTester_0.Status.staReceived AND SKTcpClientTester_0.Status.DataRecv[2]= 2 AND SKTcpClientTester_0.Status.DataRecv[5]= 3 THEN
                SKTcpClientTester_0.Cmd.Send:= FALSE;
                IF SC_OvlTesteraHV.IdleTime.Q THEN
                    SC_OvlTesteraHV.ResetStep:= TRUE;
                    SC_OvlTesteraHV.Step:= 25;
                END_IF
            ELSIF SKTcpClientTester_0.Status.staError THEN
                SKTcpClientTester_0.Cmd.Send:= FALSE;
                P3_Srobovanie.STAV.Vysledok_HV_Testu:= 'NG';
                HV_Test_UKONCENY:= TRUE;
                SC_OvlTesteraHV.ResetStep:= TRUE;
                SC_OvlTesteraHV.Step:= 100;
            END_IF

        30:
            SC_OvlTesteraHV.StepName:= '30 - Potvrdenie precitanie vysledkov testu - typ 3';
            SC_OvlTesteraHV.IdleTime.PT:= T#300ms;
            SC_OvlTesteraHV.AlarmTime.PT:= T#10s;
            SC_OvlTesteraHV.IdleTime.IN:= TRUE;

            SKTcpClientTester_0.Params.Packet.type:= 3;
            SKTcpClientTester_0.Params.Packet.workplace:= 46;
            SKTcpClientTester_0.Params.Packet.id:= 1;
            SKTcpClientTester_0.Cmd.Send:= TRUE;

            IF SKTcpClientTester_0.Cmd.Send AND NOT SKTcpClientTester_0.Status.staReceived AND NOT SKTcpClientTester_0.Status.staError THEN
                SC_OvlTesteraHV.ResetStep:= TRUE;
                SC_OvlTesteraHV.Step:= 33;
            END_IF

        33:
            SC_OvlTesteraHV.StepName:= '33 - Odpoved testera na potvrdenie vysledkov - typ 3';
            SC_OvlTesteraHV.IdleTime.PT:= T#300ms;
            SC_OvlTesteraHV.AlarmTime.PT:= T#10s;

            IF SKTcpClientTester_0.Status.staReceived AND SKTcpClientTester_0.Status.DataRecv[2]= 3 AND SKTcpClientTester_0.Status.DataRecv[5]= 0 THEN
                SKTcpClientTester_0.Cmd.Send:= FALSE;
                NameranyCas_CelkovyCasTestovania:= Cas_HVTester.ET;
                Cas_HVTester.IN:= FALSE;
                HV_Test_UKONCENY:= TRUE;
                SC_OvlTesteraHV.ResetStep:= TRUE;
                SC_OvlTesteraHV.Step:= 100;
            ELSIF SKTcpClientTester_0.Status.staReceived AND SKTcpClientTester_0.Status.DataRecv[2]= 3 AND SKTcpClientTester_0.Status.DataRecv[5]= 1 THEN
                P3_Srobovanie.STAV.Vysledok_HV_Testu:= 'NG';
                NameranyCas_CelkovyCasTestovania:= Cas_HVTester.ET;
                Cas_HVTester.IN:= FALSE;
                HV_Test_UKONCENY:= TRUE;
                SKTcpClientTester_0.Cmd.Send:= FALSE;
                SC_OvlTesteraHV.ResetStep:= TRUE;
                SC_OvlTesteraHV.Step:= 100;
            ELSIF SKTcpClientTester_0.Status.staError THEN
                SKTcpClientTester_0.Cmd.Send:= FALSE;
                SC_OvlTesteraHV.ResetStep:= TRUE;
                SC_OvlTesteraHV.Step:= 100;
            END_IF

        100:
            SC_OvlTesteraHV.StepName:= '100 - Cakam na zrusenie signalu start testovania';
            SC_OvlTesteraHV.IdleTime.PT:= T#3s;
            SC_OvlTesteraHV.AlarmTime.PT:= T#10s;

            IF NOT HV_Test_START THEN
                SC_OvlTesteraHV.ResetStep:= TRUE;
                SC_OvlTesteraHV.Step:= 0;
            END_IF

    END_CASE

END_ACTION
```

### Program Logical/Program/Pracovisko_3/P3_SkrutkovaciSet_M5 (IEC)

#### Main.st - Init, cyclic, exit code
```iecst
PROGRAM _INIT
	TprazdnyZasobnik.PT:=T#2000ms;
	TakumulaciaPlna.PT:=T#1000ms;
	TakumulaciaPrazdna.PT:=T#1000ms;
	TvytvorenieVakua.PT:=T#200ms;
	TodvetranieVakua.PT:=T#200ms;
	TvibrovanieHrniec.PT:=T#3000ms;
	TvibrovanieLista.PT:=T#3000ms;
	TpredOtocenim.PT:= T#1000ms;
	TvyfukovaniePredVibrovanim.PT:= T#1000ms;
	TvypnutieOfuku.PT:= T#2000ms;
	TpoOtoceni.PT:= T#5s;
	TofukVibrolisty.PT:= T#1000ms;
END_PROGRAM

PROGRAM _CYCLIC

	(********************Mapovanie IN/OUT********************************)
	SkrutkovaciSet.Manual:= P3_Srobovanie.SkrutkovaciSet_M5.Manual;
	SkrutkovaciSet.Automat:= P3_Srobovanie.SkrutkovaciSet_M5.Automat;
	SkrutkovaciSet.SkrutkaOdobrata:=P3_Srobovanie.SkrutkovaciSet_M5.SkrutkaM5_Odobrata;
	P3_Srobovanie.SkrutkovaciSet_M5.SkrutkaM5_Pripravena:= SkrutkovaciSet.SkrutkaPripravena;

	IF P3_Srobovanie.SkrutkovaciSet_M5.Reset THEN
		SkrutkovaciSet.VretenoFaza:=0;
		P3_Srobovanie.SkrutkovaciSet_M5.Reset:= FALSE;
	END_IF

	SkrutkovaciSet.Vreteno.IN.ReturnStroke:=P3_Srobovanie.IN.SkrutkM5_ZASUNUTY_MS57;
	SkrutkovaciSet.Vreteno.IN.VakuumDosiahnute:=P3_Srobovanie.IN.SkrutkM5_SnimacVakua_S29;

	SkrutkovaciSet.Zasobnik.IN.AccumulationSwitchStart:=P3_Srobovanie.IN.VibrolistaSrobM5_ZACIATOK_OS18;
	SkrutkovaciSet.Zasobnik.IN.AccumulationSwitchEnd:=P3_Srobovanie.IN.ZasobSrobM5_ListaPLNA_OS16;
	SkrutkovaciSet.Zasobnik.IN.EscapementPickUp:=P3_Srobovanie.IN.OddelSrobM5_OtocenyVZAD_MS55;
	SkrutkovaciSet.Zasobnik.IN.EscapementDrop:=P3_Srobovanie.IN.OddelSrobM5_OtocenyVPRED_MS56;
	SkrutkovaciSet.Zasobnik.IN.FeederLevelControl:=P3_Srobovanie.IN.ZasobSrobM5_PRAZDNY_IS83;
	SkrutkovaciSet.Zasobnik.IN.InlineControl:=P3_Srobovanie.IN.OddelSrobM5_SrobaNaVstupe_OS19;
	SkrutkovaciSet.Zasobnik.IN.ScrewAvailable:=P3_Srobovanie.IN.OddelSrobM5_SrobaNaVystupe_OS20;

	P3_Srobovanie.OUT.ZasobSrobM5_Ofuk_RUN_YV125:=SkrutkovaciSet.Zasobnik.OUT.BlowOff;
	P3_Srobovanie.OUT.OddelovacSrobM5_OtocVPRED_YV128:=SkrutkovaciSet.Zasobnik.OUT.EscapementDrop;
	P3_Srobovanie.OUT.OddelovacSrobM5_OtocVZAD_YV127:=SkrutkovaciSet.Zasobnik.OUT.EscapementPickUp;
	P3_Srobovanie.OUT.ZasobSrobM5_OfukTried_RUN_YV126:=SkrutkovaciSet.Zasobnik.OUT.SortingAir;
	P3_Srobovanie.OUT.ZasobSrobM5_Vibrovanie_RUN_FM16:=SkrutkovaciSet.Zasobnik.OUT.StartA20Hrniec;
	P3_Srobovanie.OUT.VibrolistaSrobM5_Vibrov_RUN_FM17:=SkrutkovaciSet.Zasobnik.OUT.StartA20Lista;

	(********************Časáky********************************)
	TprazdnyZasobnik();
	TakumulaciaPlna();
	TakumulaciaPrazdna();
	TvytvorenieVakua();
	TodvetranieVakua();
	TvibrovanieHrniec();
	TvibrovanieLista();
	TpredOtocenim();
	TvyfukovaniePredVibrovanim();
	TvypnutieOfuku();
	TpoOtoceni();
	TofukVibrolisty();
	(********************Zásobnik********************************)
	//kontrola akumulacie
	IF SkrutkovaciSet.Zasobnik.IN.AccumulationSwitchStart=1 THEN
		TakumulaciaPlna.IN:=1;
	ELSE
		TakumulaciaPlna.IN:=0;
	END_IF

	IF SkrutkovaciSet.Zasobnik.IN.AccumulationSwitchEnd=0 THEN
		TakumulaciaPrazdna.IN:=1;
	ELSE
		TakumulaciaPrazdna.IN:=0;
	END_IF

	//kontrola naplnenia zasobnika
	IF SkrutkovaciSet.Zasobnik.IN.FeederLevelControl=1 THEN
		TprazdnyZasobnik.IN:=1;
	ELSE
		TprazdnyZasobnik.IN:=0;
	END_IF

	//Ovládanie vzduchov zásobníka//
	IF ZapniHrniec THEN
		IF TakumulaciaPlna.Q=1 AND TakumulaciaPrazdna.Q=0  THEN
			SkrutkovaciSet.Zasobnik.OUT.BlowOff:=1;
		ELSIF TakumulaciaPrazdna.Q=1 THEN
			SkrutkovaciSet.Zasobnik.OUT.BlowOff:=0;
		END_IF
		SkrutkovaciSet.Zasobnik.OUT.SortingAir:= 1;
	ELSIF ZapniListu THEN
		TofukVibrolisty.IN:= TRUE;
		SkrutkovaciSet.Zasobnik.OUT.SortingAir:= NOT TofukVibrolisty.Q;
	ELSE
		SkrutkovaciSet.Zasobnik.OUT.BlowOff:=0;
	END_IF

	TvypnutieOfuku.IN:= NOT SkrutkovaciSet.Zasobnik.OUT.StartA20Hrniec;

	IF TvypnutieOfuku.Q THEN
		SkrutkovaciSet.Zasobnik.OUT.SortingAir:= 0;
	END_IF

	//ovladanie vibracneho podavaca
	IF SkrutkovaciSet.VretenoFaza>3 AND SkrutkovaciSet.VretenoFaza<250 THEN
		IF SkrutkovaciSet.Zasobnik.IN.AccumulationSwitchStart=0 THEN
			ZapniHrniec:=1;
		ELSIF TvibrovanieHrniec.Q=1 AND SkrutkovaciSet.Zasobnik.IN.AccumulationSwitchEnd=1 AND NOT P3_Srobovanie.RR_ZapniHrniec_M5 THEN
			ZapniHrniec:=0;
		END_IF
	END_IF

	IF ZapniHrniec THEN
		TvyfukovaniePredVibrovanim.IN:= 1;
	ELSE
		TvyfukovaniePredVibrovanim.IN:= 0;
	END_IF

	IF ZapniHrniec AND TvyfukovaniePredVibrovanim.Q THEN
		SkrutkovaciSet.Zasobnik.OUT.StartA20Lista:=1;
		SkrutkovaciSet.Zasobnik.OUT.StartA20Hrniec:=1;
	ELSE
		SkrutkovaciSet.Zasobnik.OUT.StartA20Hrniec:=0;
	END_IF

	IF SkrutkovaciSet.Zasobnik.IN.AccumulationSwitchEnd=1 THEN
		TvibrovanieHrniec.IN:=1;
	ELSE
		TvibrovanieHrniec.IN:=0;
	END_IF

	//Ovládanie vybrolišty//
	IF ZapniListu AND TofukVibrolisty.Q THEN
		SkrutkovaciSet.Zasobnik.OUT.StartA20Lista:= TRUE;
	ELSE
		SkrutkovaciSet.Zasobnik.OUT.StartA20Lista:= FALSE;
	END_IF

	IF SkrutkovaciSet.Zasobnik.IN.AccumulationSwitchStart=1 AND SkrutkovaciSet.Zasobnik.OUT.StartA20Lista=1 THEN
		TvibrovanieLista.IN:=1;
	ELSE
		TvibrovanieLista.IN:=0;
	END_IF

	IF TvibrovanieLista.Q AND NOT SkrutkovaciSet.Zasobnik.IN.EscapementPickUp AND NOT P3_Srobovanie.RR_ZapniVibrolistu_M5 AND NOT SkrutkovaciSet.Zasobnik.OUT.StartA20Hrniec THEN
		ZapniListu:= FALSE;
	END_IF

	//Zapnutie hrnca v ručnom režime//
	IF EDGEPOS(P3_Srobovanie.RR_ZapniHrniec_M5) THEN
		ZapniHrniec:= TRUE;
	END_IF
	IF EDGENEG(P3_Srobovanie.RR_ZapniHrniec_M5) THEN
		ZapniHrniec:= FALSE;
	END_IF

	//Zapnutie vybrolisty v ručnom režime//
	IF EDGEPOS(P3_Srobovanie.RR_ZapniVibrolistu_M5) THEN
		ZapniListu:= TRUE;
	END_IF

	IF EDGENEG(P3_Srobovanie.RR_ZapniVibrolistu_M5) THEN
		ZapniListu:= FALSE;
	END_IF

	//Otáčenie podavača v ručnom režime//
	IF P3_Srobovanie.RR_OtocPodavacM5_VPRED THEN
		SkrutkovaciSet.Zasobnik.OUT.EscapementPickUp:= FALSE;
		SkrutkovaciSet.Zasobnik.OUT.EscapementDrop:= TRUE;
		P3_Srobovanie.RR_OtocPodavacM5_VPRED:= FALSE;
	ELSIF P3_Srobovanie.RR_OtocPodavacM5_VZAD THEN
		SkrutkovaciSet.Zasobnik.OUT.EscapementDrop:= FALSE;
		SkrutkovaciSet.Zasobnik.OUT.EscapementPickUp:= TRUE;
		P3_Srobovanie.RR_OtocPodavacM5_VZAD:= FALSE;
	END_IF

	IF P3_Srobovanie.IN.OddelSrobM5_OtocenyVPRED_MS56 THEN
		SkrutkovaciSet.Zasobnik.OUT.EscapementDrop:= FALSE;
	END_IF

	IF P3_Srobovanie.IN.OddelSrobM5_OtocenyVZAD_MS55 THEN
		SkrutkovaciSet.Zasobnik.OUT.EscapementPickUp:= FALSE;
	END_IF

	(********************Vreteno********************************)
	CASE SkrutkovaciSet.VretenoFaza OF
		0: SkrutkovaciSet.VretenoStatus:="Vypnute";
			SkrutkovaciSet.Vreteno.OUT.Spindle:=0;
			SkrutkovaciSet.Vreteno.OUT.VacuumOff:=0;
			SkrutkovaciSet.Vreteno.OUT.VacuumOn:=0;

			SkrutkovaciSet.Zasobnik.OUT.EscapementDrop:=0;
			SkrutkovaciSet.Zasobnik.OUT.EscapementPickUp:=0;

			SkrutkovaciSet.Zasobnik.OUT.StartA20Hrniec:=0;
			SkrutkovaciSet.Zasobnik.OUT.StartA20Lista:=0;
			SkrutkovaciSet.Manual:= 0;
			SkrutkovaciSet.Automat:= 0;
			SkrutkovaciSet.SkrutkaOdobrata:= 0;
			SkrutkovaciSet.SkrutkaPripravena:= 0;
			TpredOtocenim.IN:= 0;
			TpoOtoceni.IN:= 0;
			TvyfukovaniePredVibrovanim.IN:= 0;
			TpodaniaSkrutky.IN:= 0;
			ZapniHrniec:= 0;
			ZapniListu:= 0;
			P3_Srobovanie.STAV.Podanie_M5_BUSY:= FALSE;
			SkrutkovaciSet.VretenoFaza:=1;

		1: SkrutkovaciSet.VretenoStatus:="Inicializacia: cakam na povel";
			IF SkrutkovaciSet.Automat=1 THEN
				SkrutkovaciSet.VretenoFaza:=2;
			ELSIF SkrutkovaciSet.Manual=1 THEN
				SkrutkovaciSet.VretenoFaza:=250;
			ELSIF P3_Srobovanie.RR_PodajSkrutkuM5 THEN
				P3_Srobovanie.STAV.Podanie_M5_BUSY:= TRUE;
				SkrutkovaciSet.VretenoFaza:=2;
			END_IF

		2: SkrutkovaciSet.VretenoStatus:="Inicializacia: Cakam na natocenie kolisky na vstup";
			IF SkrutkovaciSet.Zasobnik.IN.ScrewAvailable=1 THEN
				SkrutkovaciSet.VretenoFaza:=10;
			ELSE
				SkrutkovaciSet.Zasobnik.OUT.EscapementDrop:=0;
				SkrutkovaciSet.Zasobnik.OUT.EscapementPickUp:=1;
				IF SkrutkovaciSet.Zasobnik.IN.EscapementPickUp=1 THEN
					SkrutkovaciSet.VretenoFaza:=3;
				END_IF
			END_IF

		3: SkrutkovaciSet.VretenoStatus:="Inicializacia: Cakam na pritomnost skrutky na vstupe";
			ZapniListu:=1;
			ZapniHrniec:= 1;
			IF SkrutkovaciSet.Zasobnik.IN.InlineControl=1 THEN
				SkrutkovaciSet.VretenoFaza:=4;
			END_IF

		4: SkrutkovaciSet.VretenoStatus:="Inicializacia: Natocenie kolisky na vystup";
			TpredOtocenim.IN:= 1;
			IF TpredOtocenim.Q THEN
				TpredOtocenim.IN:= 0;
				SkrutkovaciSet.Zasobnik.OUT.EscapementDrop:=1;
				SkrutkovaciSet.Zasobnik.OUT.EscapementPickUp:=0;
				SkrutkovaciSet.VretenoFaza:=8;
			END_IF

		8: SkrutkovaciSet.VretenoStatus:="Inicializacia: Cakam na natocenie kolisky na vystup";
			TpoOtoceni.IN:= 1;
			IF SkrutkovaciSet.Zasobnik.IN.EscapementDrop=1 THEN
				TpoOtoceni.IN:= 0;
				SkrutkovaciSet.VretenoFaza:=10;
			ELSIF TpoOtoceni.Q THEN
				TpoOtoceni.IN:= 0;
				SkrutkovaciSet.Zasobnik.OUT.EscapementDrop:=0;
				SkrutkovaciSet.Zasobnik.OUT.EscapementPickUp:=1;
				SkrutkovaciSet.VretenoFaza:=4;
			END_IF

		10: SkrutkovaciSet.VretenoStatus:="Inicializacia: Cakam na pritomnost skrutky na vystupe";
			IF SkrutkovaciSet.Zasobnik.IN.ScrewAvailable=1 THEN
				SkrutkovaciSet.VretenoFaza:=100;
			END_IF

		100: SkrutkovaciSet.VretenoStatus:="Pripravene: cakam na povel";
			SkrutkovaciSet.SkrutkaPripravena:=1;
			IF SkrutkovaciSet.SkrutkaOdobrata=1 THEN
				SkrutkovaciSet.VretenoFaza:=101;
			ELSIF P3_Srobovanie.RR_PodajSkrutkuM5 THEN
				P3_Srobovanie.STAV.Podanie_M5_BUSY:= FALSE;
				P3_Srobovanie.RR_PodajSkrutkuM5:= FALSE;
				SkrutkovaciSet.VretenoFaza:=0;
			END_IF

		101: SkrutkovaciSet.VretenoStatus:="Cakam kym zmizne skrutka zo snimaca";

			IF SkrutkovaciSet.Zasobnik.IN.ScrewAvailable=0 THEN
				SkrutkovaciSet.SkrutkaPripravena:=0;
				SkrutkovaciSet.VretenoFaza:=102;
			END_IF

		102: SkrutkovaciSet.VretenoStatus:="Cakam na zrusenie signalu skrutka odobrata";
			IF SkrutkovaciSet.SkrutkaOdobrata=0 THEN
				SkrutkovaciSet.VretenoFaza:=150;
			END_IF

		150: SkrutkovaciSet.VretenoStatus:="Cakam na otocenie kolisky na vstup";
			SkrutkovaciSet.Zasobnik.OUT.EscapementDrop:=0;
			SkrutkovaciSet.Zasobnik.OUT.EscapementPickUp:=1;
			IF SkrutkovaciSet.Zasobnik.IN.EscapementPickUp=1 THEN
				ZapniListu:=1;
				ZapniHrniec:= 1;
				SkrutkovaciSet.VretenoFaza:=151;
			END_IF

		151: SkrutkovaciSet.VretenoStatus:="Inicializacia: Cakam na pritomnost skrutky na vstupe";
			IF SkrutkovaciSet.Zasobnik.IN.InlineControl=1 THEN
				SkrutkovaciSet.VretenoFaza:=152;
			END_IF

		152: SkrutkovaciSet.VretenoStatus:="Inicializacia: Natocenie kolisky na vystup";
			TpredOtocenim.IN:= 1;
			IF TpredOtocenim.Q THEN
				TpredOtocenim.IN:= 0;
				SkrutkovaciSet.Zasobnik.OUT.EscapementDrop:=1;
				SkrutkovaciSet.Zasobnik.OUT.EscapementPickUp:=0;
				SkrutkovaciSet.VretenoFaza:=153;
			END_IF

		153: SkrutkovaciSet.VretenoStatus:="Inicializacia: Cakam na natocenie kolisky na vystup";
			TpoOtoceni.IN:= 1;
			IF SkrutkovaciSet.Zasobnik.IN.EscapementDrop=1 THEN
				TpoOtoceni.IN:= 0;
				SkrutkovaciSet.VretenoFaza:=155;
			ELSIF TpoOtoceni.Q THEN
				TpoOtoceni.IN:= 0;
				SkrutkovaciSet.Zasobnik.OUT.EscapementDrop:=0;
				SkrutkovaciSet.Zasobnik.OUT.EscapementPickUp:=1;
				SkrutkovaciSet.VretenoFaza:=152;
			END_IF

		155: SkrutkovaciSet.VretenoStatus:="Inicializacia: Cakam na pritomnost skrutky na vystupe";
			IF SkrutkovaciSet.Zasobnik.IN.ScrewAvailable=1 THEN
				SkrutkovaciSet.VretenoFaza:=100;
			END_IF

		250: SkrutkovaciSet.VretenoStatus:="Rucny rezim";
			SkrutkovaciSet.Manual:=0;
	END_CASE

END_PROGRAM

PROGRAM _EXIT
END_PROGRAM
```

#### Types.typ - Local data types
```iecst
TYPE
	SkrutkovaciSetStruc : 	STRUCT
		VretenoStatus : WSTRING[80];
		VretenoFaza : USINT;
		Zasobnik : ZasobnikStruc;
		Vreteno : VretenoStruc;
		SkrutkaOdobrata : BOOL;
		SkrutkaPripravena : BOOL;
		Manual : BOOL;
		Automat : BOOL;
	END_STRUCT;
	INzasobnik : 	STRUCT
		AccumulationSwitchEnd : BOOL; (*Snimac zaplnenia listy koniec S28*)
		AccumulationSwitchStart : BOOL; (*Snimac zaplnenia zaciatok listy S25*)
		EscapementDrop : BOOL; (*Koliska na odoberani skrutky S22*)
		EscapementPickUp : BOOL; (*Koliska na naberani skrutky S23*)
		InlineControl : BOOL; (*Srobka v koliske S24*)
		ScrewAvailable : BOOL; (*Srobka na odoberani S21*)
		FeederLevelControl : BOOL; (*Hladina v zasobniku S20*)
	END_STRUCT;
	OUTzasobnik : 	STRUCT
		StartA20Lista : BOOL; (*Zapnutie vibrovania A20 na liste*)
		StartA20Hrniec : BOOL; (*Zapnutie vibrovania A20 v hrnci*)
		EscapementDrop : BOOL; (*Koliska na odoberanie Y22*)
		EscapementPickUp : BOOL; (*Koliska na naberanie Y23*)
		SortingAir : BOOL; (*Triedenie kusov Y30*)
		BlowOff : BOOL; (*Zhadzovanie kusov Y25*)
	END_STRUCT;
	INvreteno : 	STRUCT
		VretenoVysunuteSrobovanie : BOOL; (*IOlink signal*)
		VretenoVysunuteOdhadzovanie : BOOL; (*IOlink signal*)
		VretenoVysunuteOdoberanie : BOOL; (*IOlink signal*)
		VakuumDosiahnute : BOOL; (*Vakuum dosiahnute S28*)
		ReturnStroke : BOOL; (*Vreteno zasunute S01*)
	END_STRUCT;
	OUTvreteno : 	STRUCT
		Spindle : BOOL; (*Vysunutie vretena Y02*)
		VacuumOff : BOOL; (*Vypnutie vakua na pridrzanie skrutky Y15*)
		VacuumOn : BOOL; (*Pridrzanie skrutky Y15*)
	END_STRUCT;
	VretenoStruc : 	STRUCT
		OUT : OUTvreteno;
		IN : INvreteno;
	END_STRUCT;
	ZasobnikStruc : 	STRUCT
		OUT : OUTzasobnik;
		IN : INzasobnik;
	END_STRUCT;
END_TYPE
```

#### Variables.var - Local variables
```iecst
VAR
	SkrutkovaciSet : SkrutkovaciSetStruc;
	TprazdnyZasobnik : TON;
	TakumulaciaPrazdna : TON;
	TakumulaciaPlna : TON;
	TvytvorenieVakua : TON;
	TodvetranieVakua : TON;
	TvibrovanieLista : TON;
	TvibrovanieHrniec : TON;
	TpredOtocenim : TON;
	TvyfukovaniePredVibrovanim : TON;
	ZapniHrniec : BOOL;
	ZapniListu : BOOL;
	TpodaniaSkrutky : TON;
	TvypnutieOfuku : TON;
	TpoOtoceni : TON;
	TofukVibrolisty : TON;
END_VAR
```

### Program Logical/Program/Pracovisko_3/P3_SkrutkovaciSet_K40 (IEC)
